C01819=1087.779,-102.417,-50.994,174.374,16.859,152.716
C01820=1087.774,-102.667,-50.984,174.373,16.858,152.716
C01821=1087.768,-102.917,-50.974,174.371,16.857,152.716
C01822=1087.761,-103.166,-50.965,174.369,16.856,152.716
C01823=1087.755,-103.416,-50.955,174.368,16.856,152.716
C01824=1087.749,-103.666,-50.944,174.367,16.855,152.716
C01825=1087.743,-103.916,-50.935,174.365,16.854,152.716
C01826=1087.737,-104.165,-50.925,174.363,16.853,152.717
C01827=1087.731,-104.415,-50.915,174.362,16.852,152.717
C01828=1087.724,-104.664,-50.905,174.361,16.851,152.717
C01829=1087.719,-104.914,-50.895,174.359,16.851,152.717
C01830=1087.713,-105.164,-50.886,174.357,16.850,152.717
C01831=1087.707,-105.414,-50.876,174.355,16.849,152.717
C01832=1087.700,-105.663,-50.866,174.354,16.849,152.718
C01833=1087.695,-105.913,-50.856,174.353,16.847,152.718
C01834=1087.689,-106.163,-50.846,174.351,16.847,152.718
C01835=1087.682,-106.413,-50.837,174.349,16.846,152.718
C01836=1087.676,-106.663,-50.827,174.348,16.845,152.718
C01837=1087.670,-106.912,-50.817,174.347,16.845,152.718
C01838=1087.664,-107.162,-50.807,174.345,16.844,152.718
C01839=1087.658,-107.412,-50.797,174.343,16.842,152.719
C01840=1087.652,-107.662,-50.787,174.342,16.842,152.719
C01841=1087.646,-107.911,-50.778,174.341,16.841,152.719
C01842=1087.640,-108.161,-50.768,174.339,16.841,152.719
C01843=1087.633,-108.411,-50.759,174.337,16.840,152.719
C01844=1087.627,-108.660,-50.748,174.336,16.840,152.719
C01845=1087.621,-108.910,-50.739,174.334,16.839,152.720
C01846=1087.615,-109.160,-50.729,174.333,16.837,152.720
C01847=1087.609,-109.410,-50.719,174.331,16.837,152.720
C01848=1087.603,-109.660,-50.710,174.330,16.836,152.720
C01849=1087.597,-109.909,-50.700,174.328,16.836,152.720
C01850=1087.591,-110.159,-50.691,174.326,16.835,152.720
C01851=1087.585,-110.408,-50.681,174.324,16.834,152.721
C01852=1087.579,-110.658,-50.672,174.324,16.833,152.721
C01853=1087.573,-110.908,-50.662,174.322,16.833,152.721
C01854=1087.567,-111.158,-50.653,174.320,16.832,152.721
C01855=1087.560,-111.407,-50.642,174.318,16.831,152.721
C01856=1087.554,-111.657,-50.633,174.317,16.831,152.721
C01857=1087.548,-111.907,-50.623,174.315,16.830,152.722
C01858=1087.542,-112.156,-50.614,174.314,16.829,152.722
C01859=1087.535,-112.406,-50.604,174.313,16.829,152.722
C01860=1087.529,-112.656,-50.594,174.311,16.828,152.722
C01861=1087.523,-112.927,-50.584,174.309,16.827,152.722
C01862=1087.517,-113.198,-50.574,174.307,16.826,152.723
C01863=1087.510,-113.469,-50.563,174.306,16.826,152.723
C01864=1087.503,-113.741,-50.553,174.304,16.824,152.723
C01865=1087.497,-113.991,-50.543,174.303,16.824,152.723
C01866=1087.491,-114.240,-50.534,174.301,16.823,152.723
C01867=1087.485,-114.490,-50.524,174.299,16.823,152.724
C01868=1087.479,-114.740,-50.515,174.298,16.822,152.724
C01869=1087.473,-114.989,-50.505,174.296,16.822,152.724
C01870=1087.467,-115.239,-50.496,174.295,16.821,152.724
C01871=1087.461,-115.489,-50.486,174.293,16.820,152.724
C01872=1087.454,-115.738,-50.477,174.292,16.819,152.724
C01873=1087.448,-115.988,-50.467,174.290,16.819,152.725
C01874=1087.442,-116.238,-50.458,174.288,16.818,152.725
C01875=1087.436,-116.488,-50.448,174.287,16.818,152.725
C01876=1087.430,-116.738,-50.438,174.286,16.817,152.725
C01877=1087.424,-116.987,-50.429,174.284,16.816,152.725
C01878=1087.418,-117.238,-50.420,174.282,16.815,152.726
C01879=1087.412,-117.487,-50.411,174.281,16.815,152.726
C01880=1087.406,-117.737,-50.401,174.279,16.814,152.726
C01881=1087.399,-117.986,-50.392,174.277,16.814,152.726
C01882=1087.393,-118.236,-50.383,174.276,16.813,152.726
C01883=1087.387,-118.486,-50.373,174.275,16.813,152.726
C01884=1087.381,-118.736,-50.364,174.273,16.812,152.727
C01885=1087.374,-118.985,-50.354,174.272,16.811,152.727
C01886=1087.368,-119.235,-50.344,174.270,16.811,152.727
C01887=1087.363,-119.484,-50.335,174.268,16.810,152.727
C01888=1087.357,-119.735,-50.326,174.267,16.810,152.727
C01889=1087.351,-119.985,-50.317,174.265,16.809,152.728
C01890=1087.344,-120.234,-50.308,174.264,16.808,152.728
C01891=1087.338,-120.484,-50.298,174.262,16.808,152.728
C01892=1087.331,-120.734,-50.289,174.261,16.807,152.728
C01893=1087.325,-120.983,-50.279,174.259,16.806,152.728
C01894=1087.320,-121.233,-50.271,174.257,16.806,152.729
C01895=1087.314,-121.483,-50.261,174.256,16.806,152.729
C01896=1087.308,-121.733,-50.252,174.254,16.805,152.729
C01897=1087.301,-121.982,-50.243,174.252,16.804,152.729
C01898=1087.295,-122.232,-50.233,174.251,16.804,152.729
C01899=1087.288,-122.482,-50.223,174.250,16.803,152.730
C01900=1087.283,-122.732,-50.215,174.248,16.802,152.730
C01901=1087.277,-122.981,-50.205,174.247,16.802,152.730
C01902=1087.271,-123.231,-50.196,174.245,16.801,152.730
C01903=1087.264,-123.481,-50.187,174.243,16.801,152.730
C01904=1087.258,-123.731,-50.178,174.242,16.801,152.731
C01905=1087.252,-123.981,-50.168,174.240,16.800,152.731
C01906=1087.246,-124.230,-50.159,174.238,16.799,152.731
C01907=1087.240,-124.480,-50.150,174.237,16.799,152.731
C01908=1087.234,-124.730,-50.141,174.236,16.798,152.731
C01909=1087.227,-124.980,-50.132,174.234,16.797,152.732
C01910=1087.221,-125.229,-50.122,174.233,16.797,152.732
C01911=1087.216,-125.479,-50.113,174.231,16.797,152.732
C01912=1087.209,-125.729,-50.105,174.229,16.796,152.732
C01913=1087.203,-125.978,-50.095,174.228,16.796,152.732
C01914=1087.197,-126.228,-50.086,174.226,16.795,152.733
C01915=1087.190,-126.478,-50.076,174.225,16.795,152.733
C01916=1087.184,-126.728,-50.068,174.223,16.794,152.733
C01917=1087.178,-126.977,-50.059,174.221,16.793,152.733
C01918=1087.172,-127.227,-50.049,174.220,16.793,152.734
C01919=1087.165,-127.477,-50.041,174.218,16.793,152.734
C01920=1087.159,-127.727,-50.031,174.216,16.792,152.734
C01921=1087.153,-127.984,-50.022,174.215,16.792,152.734
C01922=1087.148,-128.242,-50.012,174.214,16.790,152.734
C01923=1087.150,-128.498,-50.000,174.213,16.788,152.734
C01924=1087.156,-128.753,-49.987,174.213,16.784,152.733
C01925=1086.753,-128.774,-50.114,174.170,16.892,152.762
C01926=1086.746,-128.521,-50.128,174.171,16.896,152.763
C01927=1086.745,-128.264,-50.139,174.172,16.899,152.763
C01928=1086.750,-128.006,-50.150,174.173,16.900,152.763
C01929=1086.756,-127.749,-50.159,174.175,16.900,152.763
C01930=1086.762,-127.499,-50.167,174.177,16.901,152.763
C01931=1086.768,-127.249,-50.177,174.178,16.901,152.762
C01932=1086.774,-126.999,-50.187,174.180,16.902,152.762
C01933=1086.780,-126.750,-50.194,174.181,16.903,152.762
C01934=1086.786,-126.500,-50.204,174.182,16.903,152.762
C01935=1086.792,-126.250,-50.214,174.184,16.904,152.762
C01936=1086.799,-126.000,-50.222,174.186,16.904,152.761
C01937=1086.805,-125.750,-50.231,174.187,16.904,152.761
C01938=1086.811,-125.501,-50.241,174.189,16.905,152.761
C01939=1086.817,-125.252,-50.250,174.191,16.906,152.761
C01940=1086.823,-125.001,-50.258,174.192,16.906,152.760
C01941=1086.830,-124.752,-50.268,174.194,16.907,152.760
C01942=1086.836,-124.502,-50.278,174.195,16.908,152.760
C01943=1086.842,-124.252,-50.287,174.197,16.908,152.760
C01944=1086.847,-124.002,-50.296,174.198,16.909,152.760
C01945=1086.854,-123.753,-50.305,174.200,16.909,152.760
C01946=1086.860,-123.503,-50.314,174.201,16.909,152.759
C01947=1086.866,-123.253,-50.324,174.203,16.910,152.759
C01948=1086.873,-123.003,-50.333,174.205,16.911,152.759
C01949=1086.878,-122.754,-50.342,174.206,16.911,152.759
C01950=1086.885,-122.504,-50.351,174.208,16.912,152.759
C01951=1086.891,-122.254,-50.360,174.209,16.913,152.758
C01952=1086.897,-122.005,-50.370,174.211,16.913,152.758
C01953=1086.903,-121.755,-50.379,174.212,16.914,152.758
C01954=1086.909,-121.504,-50.388,174.214,16.914,152.758
C01955=1086.915,-121.255,-50.398,174.215,16.914,152.758
C01956=1086.921,-121.005,-50.407,174.217,16.915,152.757
C01957=1086.928,-120.756,-50.416,174.219,16.916,152.757
C01958=1086.934,-120.506,-50.426,174.220,16.917,152.757
C01959=1086.940,-120.256,-50.435,174.222,16.917,152.757
C01960=1086.946,-120.006,-50.444,174.223,16.918,152.757
C01961=1086.952,-119.756,-50.454,174.224,16.918,152.756
C01962=1086.958,-119.507,-50.463,174.226,16.919,152.756
C01963=1086.964,-119.257,-50.472,174.228,16.920,152.756
C01964=1086.970,-119.008,-50.482,174.230,16.921,152.756
C01965=1086.977,-118.758,-50.491,174.231,16.921,152.756
C01966=1086.983,-118.508,-50.500,174.232,16.922,152.755
C01967=1086.989,-118.258,-50.510,174.234,16.922,152.755
C01968=1086.995,-118.008,-50.519,174.235,16.923,152.755
C01969=1087.001,-117.758,-50.528,174.237,16.923,152.755
C01970=1087.007,-117.509,-50.538,174.239,16.924,152.755
C01971=1087.013,-117.259,-50.547,174.240,16.924,152.755
C01972=1087.019,-117.010,-50.557,174.242,16.925,152.754
C01973=1087.025,-116.760,-50.566,174.243,16.926,152.754
C01974=1087.032,-116.510,-50.576,174.245,16.927,152.754
C01975=1087.038,-116.260,-50.586,174.246,16.927,152.754
C01976=1087.044,-116.010,-50.595,174.248,16.928,152.754
C01977=1087.050,-115.761,-50.605,174.250,16.929,152.753
C01978=1087.056,-115.511,-50.614,174.251,16.929,152.753
C01979=1087.062,-115.262,-50.623,174.253,16.930,152.753
C01980=1087.069,-115.012,-50.632,174.254,16.931,152.753
C01981=1087.075,-114.762,-50.642,174.256,16.932,152.753
C01982=1087.081,-114.513,-50.652,174.257,16.932,152.753
C01983=1087.087,-114.263,-50.661,174.259,16.933,152.752
C01984=1087.094,-114.013,-50.671,174.261,16.933,152.752
C01985=1087.099,-113.763,-50.681,174.262,16.934,152.752
C01986=1087.106,-113.491,-50.691,174.263,16.935,152.752
C01987=1087.112,-113.220,-50.701,174.265,16.936,152.752
C01988=1087.119,-112.948,-50.712,174.267,16.936,152.751
C01989=1087.125,-112.677,-50.722,174.269,16.937,152.751
C01990=1087.131,-112.427,-50.732,174.271,16.938,152.751
C01991=1087.138,-112.177,-50.741,174.271,16.938,152.751
C01992=1087.144,-111.927,-50.751,174.273,16.939,152.751
C01993=1087.150,-111.677,-50.760,174.275,16.940,152.751
C01994=1087.156,-111.428,-50.770,174.277,16.941,152.750
C01995=1087.162,-111.178,-50.779,174.278,16.941,152.750
C01996=1087.168,-110.928,-50.789,174.279,16.942,152.750
C01997=1087.174,-110.680,-50.799,174.281,16.943,152.750
C01998=1087.181,-110.430,-50.808,174.283,16.944,152.750
C01999=1087.187,-110.180,-50.818,174.284,16.944,152.750
C02000=1087.193,-109.930,-50.828,174.286,16.945,152.749
C02001=1087.199,-109.680,-50.837,174.288,16.946,152.749
C02002=1087.205,-109.431,-50.847,174.289,16.947,152.749
C02003=1087.211,-109.180,-50.857,174.290,16.947,152.749
C02004=1087.217,-108.931,-50.866,174.292,16.948,152.749
C02005=1087.223,-108.681,-50.876,174.294,16.949,152.749
C02006=1087.229,-108.431,-50.886,174.296,16.950,152.748
C02007=1087.236,-108.182,-50.896,174.296,16.950,152.748
C02008=1087.242,-107.932,-50.905,174.298,16.951,152.748
C02009=1087.248,-107.682,-50.915,174.300,16.952,152.748
C02010=1087.254,-107.433,-50.925,174.302,16.953,152.748
C02011=1087.260,-107.183,-50.934,174.302,16.953,152.748
C02012=1087.266,-106.933,-50.944,174.304,16.954,152.748
C02013=1087.272,-106.683,-50.955,174.306,16.955,152.747
C02014=1087.278,-106.434,-50.964,174.308,16.956,152.747
C02015=1087.285,-106.184,-50.974,174.309,16.956,152.747
C02016=1087.291,-105.934,-50.983,174.310,16.957,152.747
C02017=1087.296,-105.684,-50.993,174.312,16.958,152.747
C02018=1087.302,-105.434,-51.003,174.314,16.959,152.747
C02019=1087.309,-105.185,-51.013,174.315,16.960,152.746
C02020=1087.315,-104.935,-51.023,174.316,16.961,152.746
C02021=1087.321,-104.685,-51.032,174.318,16.961,152.746
C02022=1087.327,-104.435,-51.043,174.320,16.962,152.746
C02023=1087.333,-104.185,-51.052,174.321,16.963,152.746
C02024=1087.339,-103.936,-51.062,174.323,16.963,152.746
C02025=1087.345,-103.686,-51.072,174.324,16.964,152.746
C02026=1087.351,-103.436,-51.082,174.326,16.966,152.745
C02027=1087.357,-103.187,-51.092,174.328,16.967,152.745
C02028=1087.364,-102.937,-51.102,174.329,16.967,152.745
C02029=1087.370,-102.688,-51.112,174.330,16.968,152.745
C02030=1087.375,-102.437,-51.122,174.332,16.969,152.745
C02031=1087.382,-102.188,-51.132,174.334,16.969,152.745
C02032=1087.388,-101.938,-51.142,174.335,16.971,152.745
C02033=1087.394,-101.689,-51.151,174.337,16.972,152.744
C02034=1087.399,-101.439,-51.161,174.338,16.972,152.744
C02035=1087.406,-101.189,-51.172,174.340,16.973,152.744
C02036=1087.412,-100.940,-51.181,174.341,16.974,152.744
C02037=1087.417,-100.690,-51.191,174.343,16.975,152.744
C02038=1087.424,-100.440,-51.202,174.345,16.976,152.744
C02039=1087.430,-100.191,-51.211,174.346,16.976,152.744
C02040=1087.436,-99.941,-51.221,174.347,16.977,152.743
C02041=1087.442,-99.691,-51.232,174.349,16.978,152.743
C02042=1087.448,-99.441,-51.241,174.351,16.979,152.743
C02043=1087.454,-99.192,-51.251,174.353,16.980,152.743
C02044=1087.460,-98.942,-51.262,174.353,16.980,152.743
C02045=1087.467,-98.692,-51.272,174.355,16.982,152.743
C02046=1087.473,-98.442,-51.281,174.357,16.983,152.743
C02047=1087.479,-98.192,-51.292,174.358,16.984,152.743
C02048=1087.485,-97.943,-51.302,174.360,16.984,152.742
C02049=1087.491,-97.693,-51.312,174.361,16.985,152.742
C02050=1087.498,-97.416,-51.323,174.363,16.986,152.742
C02051=1087.504,-97.139,-51.334,174.364,16.987,152.742
C02052=1087.511,-96.863,-51.346,174.366,16.988,152.742
C02053=1087.517,-96.586,-51.356,174.368,16.989,152.742
C02054=1087.523,-96.336,-51.367,174.370,16.990,152.742
C02055=1087.529,-96.087,-51.377,174.371,16.991,152.741
C02056=1087.535,-95.837,-51.386,174.373,16.992,152.741
C02057=1087.541,-95.587,-51.397,174.375,16.993,152.741
C02058=1087.548,-95.337,-51.407,174.376,16.994,152.741
C02059=1087.554,-95.087,-51.418,174.377,16.995,152.741
C02060=1087.560,-94.838,-51.428,174.379,16.996,152.741
C02061=1087.565,-94.588,-51.438,174.380,16.997,152.741
C02062=1087.572,-94.338,-51.448,174.382,16.998,152.741
C02063=1087.577,-94.088,-51.458,174.384,16.999,152.741
C02064=1087.584,-93.839,-51.469,174.385,17.000,152.740
C02065=1087.589,-93.589,-51.479,174.386,17.000,152.740
C02066=1087.596,-93.340,-51.489,174.388,17.001,152.740
C02067=1087.601,-93.090,-51.499,174.390,17.002,152.740
C02068=1087.607,-92.841,-51.509,174.391,17.004,152.740
C02069=1087.613,-92.590,-51.520,174.393,17.005,152.740
C02070=1087.619,-92.341,-51.531,174.394,17.006,152.740
C02071=1087.625,-92.090,-51.540,174.396,17.007,152.740
C02072=1087.631,-91.841,-51.551,174.397,17.007,152.740
C02073=1087.637,-91.591,-51.561,174.399,17.008,152.739
C02074=1087.643,-91.342,-51.572,174.400,17.010,152.739
C02075=1087.649,-91.092,-51.581,174.402,17.011,152.739
C02076=1087.655,-90.842,-51.592,174.403,17.012,152.739
C02077=1087.661,-90.593,-51.602,174.405,17.013,152.739
C02078=1087.667,-90.343,-51.613,174.407,17.013,152.739
C02079=1087.674,-90.093,-51.623,174.408,17.014,152.739
C02080=1087.679,-89.843,-51.633,174.410,17.015,152.739
C02081=1087.686,-89.594,-51.644,174.411,17.016,152.738
C02082=1087.691,-89.344,-51.654,174.413,17.017,152.738
C02083=1087.697,-89.094,-51.665,174.414,17.018,152.738
C02084=1087.704,-88.845,-51.675,174.416,17.019,152.738
C02085=1087.709,-88.595,-51.685,174.418,17.021,152.738
C02086=1087.716,-88.345,-51.696,174.419,17.021,152.738
C02087=1087.721,-88.095,-51.706,174.420,17.022,152.738
C02088=1087.728,-87.846,-51.716,174.422,17.023,152.738
C02089=1087.734,-87.596,-51.727,174.423,17.024,152.738
C02090=1087.739,-87.346,-51.737,174.425,17.025,152.737
C02091=1087.746,-87.097,-51.748,174.427,17.027,152.737
C02092=1087.752,-86.847,-51.759,174.428,17.028,152.737
C02093=1087.758,-86.597,-51.768,174.430,17.029,152.737
C02094=1087.764,-86.348,-51.779,174.431,17.029,152.737
C02095=1087.770,-86.098,-51.790,174.432,17.030,152.737
C02096=1087.776,-85.848,-51.800,174.434,17.031,152.737
C02097=1087.782,-85.598,-51.811,174.436,17.033,152.737
C02098=1087.789,-85.349,-51.821,174.437,17.034,152.737
C02099=1087.794,-85.099,-51.831,174.439,17.035,152.737
C02100=1087.800,-84.849,-51.842,174.441,17.036,152.736
C02101=1087.806,-84.600,-51.853,174.442,17.037,152.736
C02102=1087.813,-84.350,-51.864,174.443,17.037,152.736
C02103=1087.819,-84.100,-51.873,174.445,17.039,152.736
C02104=1087.824,-83.851,-51.884,174.446,17.040,152.736
C02105=1087.830,-83.601,-51.895,174.448,17.041,152.736
C02106=1087.837,-83.351,-51.905,174.450,17.042,152.736
C02107=1087.843,-83.101,-51.916,174.451,17.043,152.736
C02108=1087.849,-82.852,-51.926,174.453,17.044,152.736
C02109=1087.855,-82.603,-51.937,174.455,17.045,152.735
C02110=1087.861,-82.352,-51.948,174.456,17.046,152.735
C02111=1087.867,-82.103,-51.958,174.457,17.047,152.735
C02112=1087.873,-81.853,-51.969,174.459,17.048,152.735
C02113=1087.879,-81.604,-51.980,174.460,17.049,152.735
C02114=1087.886,-81.329,-51.991,174.462,17.050,152.735
C02115=1087.893,-81.054,-52.003,174.464,17.051,152.735
C02116=1087.899,-80.779,-52.015,174.466,17.053,152.735
C02117=1087.906,-80.505,-52.026,174.467,17.054,152.735
C02118=1087.913,-80.255,-52.037,174.469,17.055,152.735
C02119=1087.918,-80.005,-52.048,174.470,17.056,152.735
C02120=1087.924,-79.756,-52.059,174.472,17.057,152.734
C02121=1087.931,-79.507,-52.069,174.473,17.058,152.734
C02122=1087.937,-79.257,-52.080,174.475,17.059,152.734
C02123=1087.942,-79.006,-52.090,174.476,17.060,152.734
C02124=1087.948,-78.757,-52.101,174.478,17.061,152.734
C02125=1087.954,-78.507,-52.112,174.480,17.063,152.734
C02126=1087.961,-78.258,-52.123,174.481,17.064,152.734
C02127=1087.967,-78.008,-52.134,174.483,17.065,152.734
C02128=1087.972,-77.759,-52.145,174.484,17.066,152.734
C02129=1087.978,-77.509,-52.155,174.486,17.067,152.734
C02130=1087.984,-77.259,-52.167,174.488,17.069,152.733
C02131=1087.990,-77.009,-52.177,174.489,17.070,152.733
C02132=1087.996,-76.759,-52.188,174.490,17.070,152.733
C02133=1088.002,-76.510,-52.198,174.491,17.072,152.733
C02134=1088.008,-76.260,-52.209,174.493,17.073,152.733
C02135=1088.014,-76.010,-52.220,174.495,17.074,152.733
C02136=1088.020,-75.761,-52.231,174.496,17.075,152.733
C02137=1088.026,-75.512,-52.242,174.498,17.076,152.733
C02138=1088.032,-75.261,-52.253,174.500,17.077,152.733
C02139=1088.038,-75.012,-52.263,174.501,17.079,152.733
C02140=1088.044,-74.763,-52.274,174.503,17.080,152.733
C02141=1088.051,-74.512,-52.285,174.504,17.081,152.733
C02142=1088.056,-74.263,-52.296,174.506,17.082,152.733
C02143=1088.062,-74.013,-52.307,174.508,17.083,152.732
C02144=1088.068,-73.763,-52.318,174.509,17.085,152.732
C02145=1088.074,-73.514,-52.329,174.511,17.086,152.732
C02146=1088.080,-73.264,-52.340,174.512,17.087,152.732
C02147=1088.086,-73.015,-52.351,174.514,17.088,152.732
C02148=1088.092,-72.765,-52.362,174.515,17.090,152.732
C02149=1088.098,-72.515,-52.373,174.517,17.091,152.732
C02150=1088.103,-72.266,-52.384,174.518,17.091,152.732
C02151=1088.109,-72.016,-52.395,174.519,17.093,152.732
C02152=1088.115,-71.766,-52.406,174.521,17.094,152.732
C02153=1088.121,-71.516,-52.417,174.522,17.095,152.732
C02154=1088.126,-71.267,-52.429,174.524,17.096,152.732
C02155=1088.132,-71.017,-52.439,174.525,17.098,152.732
C02156=1088.138,-70.767,-52.451,174.527,17.099,152.732
C02157=1088.144,-70.518,-52.462,174.529,17.100,152.732
C02158=1088.150,-70.268,-52.472,174.530,17.102,152.732
C02159=1088.156,-70.018,-52.484,174.532,17.103,152.731
C02160=1088.162,-69.768,-52.495,174.533,17.104,152.731
C02161=1088.168,-69.519,-52.505,174.535,17.105,152.731
C02162=1088.174,-69.269,-52.517,174.536,17.107,152.731
C02163=1088.180,-69.019,-52.528,174.538,17.108,152.731
C02164=1088.186,-68.770,-52.539,174.539,17.109,152.731
C02165=1088.192,-68.520,-52.550,174.541,17.110,152.731
C02166=1088.197,-68.270,-52.562,174.542,17.111,152.731
C02167=1088.203,-68.021,-52.573,174.544,17.113,152.731
C02168=1088.209,-67.771,-52.584,174.545,17.114,152.731
C02169=1088.215,-67.521,-52.595,174.547,17.115,152.731
C02170=1088.221,-67.272,-52.606,174.549,17.116,152.731
C02171=1088.227,-67.021,-52.617,174.550,17.118,152.731
C02172=1088.233,-66.773,-52.629,174.552,17.119,152.731
C02173=1088.239,-66.523,-52.639,174.553,17.120,152.731
C02174=1088.245,-66.273,-52.651,174.555,17.122,152.731
C02175=1088.250,-66.023,-52.662,174.556,17.123,152.730
C02176=1088.256,-65.774,-52.673,174.558,17.124,152.730
C02177=1088.262,-65.524,-52.685,174.559,17.126,152.730
C02178=1088.269,-65.251,-52.696,174.561,17.127,152.730
C02179=1088.275,-64.979,-52.709,174.563,17.128,152.730
C02180=1088.282,-64.707,-52.721,174.564,17.129,152.730
C02181=1088.288,-64.434,-52.734,174.566,17.131,152.730
C02182=1088.294,-64.185,-52.745,174.567,17.131,152.730
C02183=1088.300,-63.935,-52.756,174.569,17.133,152.730
C02184=1088.306,-63.686,-52.767,174.570,17.134,152.730
C02185=1088.311,-63.436,-52.779,174.572,17.135,152.730
C02186=1088.318,-63.186,-52.790,174.573,17.137,152.730
C02187=1088.323,-62.936,-52.801,174.575,17.138,152.730
C02188=1088.330,-62.687,-52.813,174.577,17.139,152.730
C02189=1088.336,-62.437,-52.824,174.578,17.141,152.730
C02190=1088.342,-62.188,-52.835,174.580,17.142,152.730
C02191=1088.347,-61.938,-52.847,174.582,17.143,152.729
C02192=1088.353,-61.688,-52.858,174.583,17.145,152.730
C02193=1088.360,-61.438,-52.869,174.585,17.146,152.729
C02194=1088.366,-61.189,-52.881,174.587,17.147,152.729
C02195=1088.372,-60.939,-52.892,174.588,17.149,152.729
C02196=1088.378,-60.690,-52.903,174.590,17.150,152.729
C02197=1088.383,-60.439,-52.915,174.591,17.152,152.729
C02198=1088.389,-60.190,-52.927,174.593,17.153,152.729
C02199=1088.396,-59.940,-52.938,174.594,17.154,152.729
C02200=1088.402,-59.691,-52.949,174.596,17.155,152.729
C02201=1088.407,-59.442,-52.960,174.597,17.156,152.729
C02202=1088.413,-59.191,-52.972,174.599,17.157,152.729
C02203=1088.419,-58.942,-52.984,174.600,17.159,152.729
C02204=1088.425,-58.692,-52.995,174.602,17.160,152.729
C02205=1088.431,-58.443,-53.006,174.604,17.161,152.729
C02206=1088.437,-58.193,-53.018,174.605,17.163,152.729
C02207=1088.443,-57.943,-53.029,174.607,17.164,152.729
C02208=1088.449,-57.694,-53.041,174.608,17.166,152.729
C02209=1088.455,-57.444,-53.052,174.610,17.167,152.729
C02210=1088.462,-57.194,-53.063,174.611,17.168,152.728
C02211=1088.467,-56.945,-53.076,174.613,17.169,152.729
C02212=1088.473,-56.695,-53.087,174.614,17.170,152.728
C02213=1088.480,-56.445,-53.099,174.616,17.172,152.728
C02214=1088.486,-56.196,-53.110,174.617,17.173,152.728
C02215=1088.492,-55.946,-53.122,174.619,17.174,152.728
C02216=1088.497,-55.696,-53.133,174.620,17.176,152.728
C02217=1088.504,-55.447,-53.145,174.622,17.177,152.728
C02218=1088.510,-55.197,-53.156,174.623,17.178,152.728
C02219=1088.516,-54.947,-53.168,174.625,17.180,152.728
C02220=1088.521,-54.698,-53.179,174.626,17.181,152.728
C02221=1088.528,-54.448,-53.191,174.628,17.182,152.728
C02222=1088.533,-54.198,-53.203,174.629,17.183,152.728
C02223=1088.540,-53.949,-53.215,174.631,17.185,152.728
C02224=1088.546,-53.699,-53.226,174.632,17.186,152.728
C02225=1088.552,-53.450,-53.238,174.634,17.187,152.728
C02226=1088.558,-53.199,-53.249,174.636,17.188,152.728
C02227=1088.564,-52.950,-53.261,174.637,17.190,152.728
C02228=1088.570,-52.700,-53.272,174.639,17.191,152.728
C02229=1088.576,-52.451,-53.284,174.641,17.193,152.728
C02230=1088.582,-52.201,-53.296,174.643,17.194,152.728
C02231=1088.588,-51.951,-53.308,174.644,17.195,152.727
C02232=1088.594,-51.702,-53.319,174.646,17.197,152.727
C02233=1088.600,-51.452,-53.331,174.647,17.198,152.727
C02234=1088.607,-51.202,-53.343,174.649,17.200,152.727
C02235=1088.612,-50.953,-53.354,174.650,17.201,152.727
C02236=1088.618,-50.703,-53.366,174.652,17.202,152.727
C02237=1088.624,-50.453,-53.377,174.653,17.203,152.727
C02238=1088.631,-50.204,-53.389,174.655,17.205,152.727
C02239=1088.636,-49.955,-53.401,174.656,17.206,152.727
C02240=1088.641,-49.704,-53.413,174.658,17.207,152.727
C02241=1088.648,-49.455,-53.425,174.659,17.209,152.727
C02242=1088.654,-49.184,-53.438,174.661,17.210,152.727
C02243=1088.660,-48.913,-53.451,174.663,17.212,152.727
C02244=1088.667,-48.641,-53.464,174.664,17.214,152.727
C02245=1088.673,-48.371,-53.476,174.666,17.215,152.727
C02246=1088.679,-48.121,-53.489,174.667,17.216,152.727
C02247=1088.686,-47.871,-53.501,174.669,17.217,152.727
C02248=1088.691,-47.621,-53.512,174.670,17.219,152.727
C02249=1088.697,-47.372,-53.524,174.673,17.221,152.727
C02250=1088.703,-47.123,-53.536,174.674,17.222,152.727
C02251=1088.708,-46.872,-53.548,174.676,17.223,152.727
C02252=1088.714,-46.623,-53.560,174.677,17.225,152.727
C02253=1088.720,-46.373,-53.572,174.679,17.226,152.727
C02254=1088.727,-46.123,-53.584,174.680,17.228,152.727
C02255=1088.732,-45.874,-53.596,174.682,17.229,152.727
C02256=1088.738,-45.625,-53.608,174.683,17.230,152.727
C02257=1088.744,-45.375,-53.620,174.685,17.232,152.727
C02258=1088.749,-45.125,-53.632,174.686,17.233,152.727
C02259=1088.756,-44.875,-53.644,174.688,17.235,152.727
C02260=1088.761,-44.626,-53.656,174.689,17.236,152.727
C02261=1088.768,-44.377,-53.668,174.691,17.238,152.726
C02262=1088.774,-44.126,-53.680,174.693,17.239,152.726
C02263=1088.779,-43.877,-53.692,174.694,17.241,152.726
C02264=1088.786,-43.627,-53.704,174.696,17.242,152.726
C02265=1088.791,-43.378,-53.716,174.697,17.243,152.726
C02266=1088.797,-43.128,-53.727,174.699,17.244,152.726
C02267=1088.803,-42.878,-53.740,174.700,17.246,152.726
C02268=1088.808,-42.629,-53.752,174.702,17.247,152.726
C02269=1088.815,-42.379,-53.764,174.703,17.249,152.726
C02270=1088.821,-42.129,-53.776,174.705,17.250,152.726
C02271=1088.826,-41.880,-53.789,174.706,17.251,152.726
C02272=1088.833,-41.630,-53.800,174.709,17.254,152.726
C02273=1088.838,-41.380,-53.812,174.710,17.255,152.726
C02274=1088.845,-41.131,-53.824,174.712,17.256,152.726
C02275=1088.850,-40.881,-53.837,174.713,17.257,152.726
C02276=1088.856,-40.631,-53.849,174.715,17.259,152.726
C02277=1088.862,-40.383,-53.861,174.716,17.260,152.726
C02278=1088.868,-40.133,-53.873,174.718,17.262,152.726
C02279=1088.874,-39.883,-53.886,174.719,17.263,152.726
C02280=1088.881,-39.633,-53.897,174.721,17.264,152.726
C02281=1088.886,-39.383,-53.909,174.723,17.266,152.726
C02282=1088.892,-39.134,-53.922,174.724,17.268,152.726
C02283=1088.898,-38.884,-53.934,174.726,17.269,152.726
C02284=1088.904,-38.635,-53.946,174.728,17.270,152.726
C02285=1088.910,-38.385,-53.959,174.729,17.272,152.726
C02286=1088.916,-38.135,-53.971,174.731,17.273,152.726
C02287=1088.922,-37.886,-53.983,174.732,17.275,152.726
C02288=1088.928,-37.636,-53.995,174.733,17.276,152.726
C02289=1088.933,-37.386,-54.008,174.735,17.277,152.726
C02290=1088.939,-37.137,-54.020,174.737,17.279,152.726
C02291=1088.945,-36.887,-54.033,174.738,17.281,152.726
C02292=1088.951,-36.637,-54.045,174.740,17.282,152.726
C02293=1088.957,-36.388,-54.057,174.741,17.284,152.726
C02294=1088.962,-36.139,-54.069,174.743,17.285,152.726
C02295=1088.968,-35.889,-54.082,174.744,17.286,152.726
C02296=1088.974,-35.639,-54.094,174.746,17.288,152.726
C02297=1088.980,-35.390,-54.107,174.747,17.289,152.726
C02298=1088.986,-35.140,-54.119,174.750,17.291,152.726
C02299=1088.991,-34.890,-54.132,174.751,17.292,152.725
C02300=1088.998,-34.640,-54.144,174.753,17.294,152.726
C02301=1089.003,-34.391,-54.156,174.754,17.295,152.726
C02302=1089.009,-34.141,-54.168,174.756,17.297,152.725
C02303=1089.015,-33.891,-54.181,174.757,17.298,152.726
C02304=1089.021,-33.642,-54.193,174.758,17.300,152.726
C02305=1089.026,-33.392,-54.206,174.761,17.301,152.725
C02306=1089.034,-33.122,-54.219,174.762,17.303,152.725
C02307=1089.039,-32.851,-54.232,174.764,17.305,152.726
C02308=1089.046,-32.580,-54.246,174.765,17.306,152.725
C02309=1089.052,-32.309,-54.260,174.767,17.308,152.725
C02310=1089.058,-32.060,-54.272,174.769,17.309,152.725
C02311=1089.064,-31.810,-54.285,174.770,17.311,152.725
C02312=1089.069,-31.561,-54.297,174.772,17.312,152.725
C02313=1089.076,-31.311,-54.309,174.773,17.313,152.725
C02314=1089.082,-31.062,-54.322,174.776,17.315,152.725
C02315=1089.088,-30.812,-54.335,174.777,17.317,152.725
C02316=1089.094,-30.562,-54.347,174.779,17.318,152.725
C02317=1089.099,-30.313,-54.359,174.780,17.320,152.725
C02318=1089.105,-30.063,-54.372,174.782,17.321,152.725
C02319=1089.111,-29.813,-54.385,174.783,17.322,152.725
C02320=1089.117,-29.564,-54.398,174.784,17.324,152.725
C02321=1089.123,-29.314,-54.410,174.787,17.326,152.725
C02322=1089.129,-29.065,-54.423,174.788,17.327,152.725
C02323=1089.134,-28.815,-54.435,174.790,17.329,152.725
C02324=1089.140,-28.565,-54.448,174.791,17.330,152.725
C02325=1089.147,-28.316,-54.460,174.793,17.331,152.725
C02326=1089.153,-28.066,-54.473,174.794,17.333,152.725
C02327=1089.159,-27.816,-54.485,174.796,17.334,152.725
C02328=1089.164,-27.567,-54.498,174.798,17.336,152.725
C02329=1089.170,-27.317,-54.510,174.799,17.337,152.725
C02330=1089.177,-27.068,-54.523,174.801,17.339,152.725
C02331=1089.182,-26.818,-54.536,174.802,17.341,152.725
C02332=1089.188,-26.568,-54.549,174.804,17.342,152.725
C02333=1089.195,-26.319,-54.562,174.805,17.343,152.725
C02334=1089.199,-26.069,-54.575,174.807,17.345,152.725
C02335=1089.205,-25.819,-54.587,174.809,17.347,152.725
C02336=1089.211,-25.570,-54.600,174.810,17.348,152.725
C02337=1089.217,-25.320,-54.613,174.812,17.350,152.725
C02338=1089.223,-25.070,-54.626,174.813,17.351,152.725
C02339=1089.228,-24.821,-54.638,174.815,17.352,152.725
C02340=1089.235,-24.572,-54.651,174.817,17.355,152.725
C02341=1089.240,-24.322,-54.664,174.818,17.356,152.725
C02342=1089.246,-24.072,-54.676,174.820,17.357,152.725
C02343=1089.252,-23.823,-54.690,174.821,17.359,152.725
C02344=1089.258,-23.573,-54.702,174.823,17.360,152.725
C02345=1089.263,-23.324,-54.715,174.825,17.362,152.725
C02346=1089.269,-23.074,-54.728,174.826,17.364,152.725
C02347=1089.275,-22.824,-54.741,174.828,17.365,152.725
C02348=1089.281,-22.575,-54.753,174.829,17.366,152.725
C02349=1089.287,-22.325,-54.766,174.831,17.368,152.725
C02350=1089.293,-22.075,-54.779,174.832,17.370,152.725
C02351=1089.298,-21.825,-54.792,174.835,17.371,152.725
C02352=1089.305,-21.576,-54.805,174.836,17.373,152.725
C02353=1089.310,-21.327,-54.817,174.837,17.374,152.725
C02354=1089.316,-21.077,-54.831,174.839,17.375,152.725
C02355=1089.322,-20.828,-54.843,174.840,17.377,152.725
C02356=1089.328,-20.578,-54.857,174.843,17.379,152.725
C02357=1089.333,-20.328,-54.870,174.844,17.380,152.725
C02358=1089.339,-20.078,-54.882,174.846,17.382,152.725
C02359=1089.346,-19.829,-54.896,174.847,17.384,152.725
C02360=1089.351,-19.579,-54.908,174.849,17.385,152.725
C02361=1089.357,-19.330,-54.922,174.851,17.387,152.725
C02362=1089.363,-19.080,-54.935,174.852,17.388,152.725
C02363=1089.369,-18.830,-54.948,174.854,17.389,152.725
C02364=1089.374,-18.581,-54.960,174.855,17.391,152.725
C02365=1089.381,-18.332,-54.973,174.856,17.393,152.725
C02366=1089.386,-18.082,-54.986,174.858,17.394,152.725
C02367=1089.392,-17.832,-55.000,174.860,17.396,152.725
C02368=1089.398,-17.583,-55.012,174.862,17.397,152.725
C02369=1089.404,-17.333,-55.025,174.863,17.399,152.725
C02370=1089.411,-17.061,-55.040,174.865,17.400,152.725
C02371=1089.417,-16.790,-55.054,174.867,17.402,152.725
C02372=1089.423,-16.518,-55.068,174.868,17.404,152.725
C02373=1089.430,-16.247,-55.083,174.871,17.406,152.725
C02374=1089.435,-15.997,-55.095,174.872,17.407,152.725
C02375=1089.442,-15.748,-55.108,174.873,17.409,152.725
C02376=1089.447,-15.499,-55.122,174.875,17.410,152.725
C02377=1089.453,-15.249,-55.135,174.876,17.411,152.725
C02378=1089.459,-14.999,-55.148,174.879,17.414,152.725
C02379=1089.464,-14.749,-55.161,174.880,17.415,152.725
C02380=1089.471,-14.500,-55.174,174.882,17.416,152.725
C02381=1089.477,-14.251,-55.188,174.883,17.418,152.725
C02382=1089.482,-14.001,-55.201,174.885,17.419,152.724
C02383=1089.488,-13.751,-55.214,174.887,17.421,152.725
C02384=1089.494,-13.502,-55.228,174.888,17.423,152.725
C02385=1089.500,-13.252,-55.240,174.890,17.424,152.725
C02386=1089.506,-13.003,-55.254,174.891,17.425,152.725
C02387=1089.511,-12.752,-55.267,174.893,17.427,152.725
C02388=1089.517,-12.503,-55.280,174.895,17.429,152.725
C02389=1089.523,-12.253,-55.294,174.896,17.431,152.725
C02390=1089.528,-12.004,-55.306,174.898,17.432,152.724
C02391=1089.534,-11.754,-55.320,174.900,17.434,152.724
C02392=1089.540,-11.505,-55.334,174.901,17.436,152.725
C02393=1089.546,-11.256,-55.347,174.903,17.437,152.724
C02394=1089.552,-11.005,-55.360,174.904,17.438,152.724
C02395=1089.558,-10.756,-55.373,174.906,17.440,152.725
C02396=1089.563,-10.506,-55.387,174.908,17.442,152.725
C02397=1089.569,-10.257,-55.400,174.910,17.443,152.724
C02398=1089.575,-10.007,-55.414,174.911,17.445,152.724
C02399=1089.581,-9.758,-55.427,174.912,17.446,152.725
C02400=1089.587,-9.508,-55.440,174.915,17.448,152.724
C02401=1089.592,-9.258,-55.453,174.916,17.449,152.724
C02402=1089.598,-9.009,-55.467,174.918,17.451,152.724
C02403=1089.604,-8.759,-55.480,174.919,17.452,152.724
C02404=1089.610,-8.510,-55.494,174.921,17.454,152.724
C02405=1089.616,-8.261,-55.508,174.923,17.456,152.724
C02406=1089.622,-8.011,-55.520,174.924,17.457,152.724
C02407=1089.627,-7.761,-55.534,174.926,17.459,152.724
C02408=1089.633,-7.512,-55.547,174.927,17.460,152.724
C02409=1089.639,-7.262,-55.561,174.929,17.462,152.724
C02410=1089.646,-7.012,-55.575,174.931,17.463,152.724
C02411=1089.651,-6.762,-55.588,174.932,17.465,152.724
C02412=1089.657,-6.513,-55.601,174.934,17.467,152.724
C02413=1089.662,-6.263,-55.615,174.936,17.468,152.724
C02414=1089.669,-6.014,-55.628,174.938,17.470,152.724
C02415=1089.674,-5.764,-55.642,174.939,17.471,152.724
C02416=1089.680,-5.515,-55.655,174.941,17.472,152.724
C02417=1089.686,-5.266,-55.669,174.943,17.475,152.724
C02418=1089.692,-5.016,-55.683,174.944,17.476,152.724
C02419=1089.697,-4.766,-55.696,174.946,17.477,152.724
C02420=1089.704,-4.516,-55.709,174.947,17.479,152.724
C02421=1089.709,-4.267,-55.723,174.949,17.481,152.724
C02422=1089.716,-4.017,-55.736,174.951,17.482,152.724
C02423=1089.721,-3.768,-55.750,174.952,17.484,152.724
C02424=1089.727,-3.519,-55.764,174.954,17.485,152.724
C02425=1089.733,-3.269,-55.777,174.956,17.487,152.724
C02426=1089.738,-3.019,-55.791,174.958,17.489,152.724
C02427=1089.745,-2.770,-55.805,174.959,17.490,152.724
C02428=1089.750,-2.521,-55.818,174.960,17.492,152.724
C02429=1089.755,-2.271,-55.832,174.963,17.493,152.724
C02430=1089.761,-2.021,-55.846,174.964,17.495,152.724
C02431=1089.768,-1.771,-55.860,174.965,17.497,152.724
C02432=1089.773,-1.522,-55.874,174.967,17.498,152.724
C02433=1089.779,-1.272,-55.888,174.969,17.500,152.724
C02434=1089.785,-1.000,-55.902,174.971,17.501,152.724
C02435=1089.791,-0.726,-55.917,174.973,17.504,152.724
C02436=1089.797,-0.453,-55.933,174.974,17.505,152.724
C02437=1089.804,-0.179,-55.948,174.976,17.507,152.724
C02438=1089.810,0.070,-55.961,174.978,17.508,152.724
C02439=1089.815,0.320,-55.975,174.979,17.510,152.724
C02440=1089.821,0.569,-55.989,174.981,17.512,152.724
C02441=1089.827,0.819,-56.002,174.983,17.514,152.724
C02442=1089.832,1.068,-56.016,174.985,17.515,152.724
C02443=1089.838,1.318,-56.030,174.986,17.516,152.724
C02444=1089.843,1.567,-56.044,174.987,17.518,152.724
C02445=1089.850,1.817,-56.058,174.990,17.520,152.724
C02446=1089.855,2.067,-56.072,174.991,17.521,152.724
C02447=1089.861,2.316,-56.085,174.993,17.523,152.724
C02448=1089.867,2.565,-56.100,174.994,17.524,152.724
C02449=1089.872,2.815,-56.114,174.996,17.526,152.724
C02450=1089.878,3.064,-56.127,174.998,17.528,152.724
C02451=1089.884,3.314,-56.141,174.999,17.529,152.724
C02452=1089.890,3.564,-56.155,175.001,17.531,152.724
C02453=1089.895,3.814,-56.169,175.003,17.532,152.724
C02454=1089.901,4.063,-56.183,175.004,17.534,152.724
C02455=1089.907,4.312,-56.197,175.006,17.536,152.724
C02456=1089.913,4.561,-56.211,175.008,17.537,152.724
C02457=1089.919,4.812,-56.225,175.010,17.539,152.724
C02458=1089.924,5.061,-56.239,175.011,17.540,152.724
C02459=1089.930,5.311,-56.253,175.013,17.542,152.724
C02460=1089.936,5.560,-56.267,175.015,17.544,152.724
C02461=1089.942,5.809,-56.281,175.016,17.545,152.724
C02462=1089.948,6.059,-56.295,175.018,17.546,152.724
C02463=1089.953,6.309,-56.309,175.020,17.548,152.724
C02464=1089.959,6.558,-56.323,175.021,17.550,152.724
C02465=1089.965,6.807,-56.337,175.023,17.551,152.724
C02466=1089.971,7.058,-56.351,175.025,17.553,152.724
C02467=1089.977,7.307,-56.365,175.027,17.555,152.724
C02468=1089.982,7.557,-56.378,175.028,17.556,152.724
C02469=1089.988,7.805,-56.393,175.030,17.558,152.724
C02470=1089.994,8.056,-56.407,175.032,17.560,152.724
C02471=1090.000,8.305,-56.421,175.033,17.561,152.724
C02472=1090.006,8.554,-56.436,175.035,17.562,152.724
C02473=1090.011,8.804,-56.450,175.037,17.565,152.724
C02474=1090.017,9.054,-56.464,175.039,17.566,152.724
C02475=1090.023,9.303,-56.477,175.040,17.567,152.724
C02476=1090.029,9.552,-56.492,175.041,17.569,152.724
C02477=1090.035,9.803,-56.506,175.044,17.570,152.724
C02478=1090.041,10.052,-56.520,175.045,17.572,152.724
C02479=1090.046,10.301,-56.534,175.047,17.574,152.724
C02480=1090.052,10.551,-56.548,175.049,17.575,152.724
C02481=1090.058,10.800,-56.563,175.050,17.577,152.724
C02482=1090.064,11.050,-56.577,175.052,17.578,152.724
C02483=1090.069,11.300,-56.591,175.054,17.580,152.724
C02484=1090.076,11.549,-56.606,175.056,17.582,152.724
C02485=1090.082,11.798,-56.619,175.057,17.583,152.724
C02486=1090.088,12.047,-56.634,175.059,17.584,152.724
C02487=1090.094,12.298,-56.648,175.061,17.586,152.724
C02488=1090.099,12.547,-56.662,175.063,17.588,152.724
C02489=1090.105,12.796,-56.676,175.064,17.589,152.724
C02490=1090.111,13.047,-56.691,175.066,17.591,152.724
C02491=1090.117,13.295,-56.705,175.068,17.592,152.724
C02492=1090.122,13.545,-56.719,175.069,17.594,152.724
C02493=1090.129,13.795,-56.734,175.072,17.596,152.724
C02494=1090.134,14.044,-56.748,175.073,17.597,152.724
C02495=1090.141,14.294,-56.763,175.074,17.599,152.724
C02496=1090.146,14.544,-56.777,175.076,17.600,152.724
C02497=1090.152,14.792,-56.791,175.078,17.602,152.724
C02498=1090.158,15.069,-56.807,175.080,17.604,152.724
C02499=1090.165,15.343,-56.823,175.082,17.605,152.723
C02500=1090.171,15.619,-56.838,175.083,17.607,152.724
C02501=1090.177,15.894,-56.855,175.086,17.609,152.724
C02502=1090.183,16.143,-56.869,175.087,17.610,152.723
C02503=1090.189,16.393,-56.883,175.089,17.612,152.723
C02504=1090.194,16.642,-56.898,175.091,17.614,152.723
C02505=1090.200,16.891,-56.912,175.092,17.615,152.723
C02506=1090.206,17.141,-56.927,175.095,17.617,152.723
C02507=1090.212,17.391,-56.941,175.096,17.619,152.723
C02508=1090.217,17.640,-56.956,175.098,17.620,152.723
C02509=1090.223,17.890,-56.971,175.100,17.622,152.723
C02510=1090.229,18.139,-56.985,175.101,17.623,152.723
C02511=1090.235,18.389,-57.000,175.103,17.624,152.723
C02512=1090.240,18.638,-57.013,175.105,17.627,152.723
C02513=1090.246,18.887,-57.028,175.107,17.628,152.723
C02514=1090.253,19.137,-57.043,175.108,17.629,152.723
C02515=1090.257,19.387,-57.057,175.110,17.631,152.723
C02516=1090.264,19.637,-57.072,175.112,17.633,152.723
C02517=1090.269,19.886,-57.086,175.113,17.634,152.723
C02518=1090.275,20.135,-57.101,175.116,17.636,152.723
C02519=1090.281,20.385,-57.116,175.117,17.637,152.723
C02520=1090.286,20.635,-57.130,175.119,17.639,152.723
C02521=1090.293,20.884,-57.145,175.121,17.641,152.723
C02522=1090.298,21.133,-57.160,175.122,17.642,152.723
C02523=1090.304,21.382,-57.174,175.124,17.644,152.723
C02524=1090.309,21.633,-57.189,175.126,17.645,152.723
C02525=1090.315,21.882,-57.204,175.128,17.647,152.723
C02526=1090.322,22.131,-57.219,175.129,17.648,152.723
C02527=1090.327,22.381,-57.233,175.131,17.650,152.723
C02528=1090.332,22.630,-57.248,175.133,17.652,152.723
C02529=1090.338,22.880,-57.263,175.134,17.653,152.723
C02530=1090.344,23.129,-57.277,175.137,17.655,152.723
C02531=1090.350,23.379,-57.292,175.138,17.656,152.723
C02532=1090.355,23.628,-57.307,175.140,17.658,152.723
C02533=1090.361,23.877,-57.321,175.142,17.660,152.723
C02534=1090.368,24.127,-57.336,175.143,17.661,152.723
C02535=1090.372,24.377,-57.351,175.145,17.662,152.723
C02536=1090.379,24.627,-57.366,175.147,17.664,152.723
C02537=1090.384,24.876,-57.380,175.149,17.666,152.723
C02538=1090.390,25.126,-57.396,175.150,17.667,152.723
C02539=1090.396,25.374,-57.410,175.153,17.669,152.723
C02540=1090.402,25.625,-57.425,175.154,17.670,152.723
C02541=1090.407,25.874,-57.440,175.156,17.672,152.723
C02542=1090.413,26.124,-57.455,175.158,17.674,152.723
C02543=1090.419,26.373,-57.469,175.159,17.675,152.723
C02544=1090.425,26.623,-57.485,175.161,17.676,152.723
C02545=1090.431,26.872,-57.499,175.163,17.678,152.722
C02546=1090.437,27.121,-57.514,175.165,17.680,152.722
C02547=1090.442,27.371,-57.529,175.167,17.682,152.723
C02548=1090.448,27.621,-57.544,175.168,17.683,152.722
C02549=1090.454,27.870,-57.558,175.170,17.684,152.722
C02550=1090.460,28.120,-57.574,175.172,17.686,152.722
C02551=1090.465,28.369,-57.588,175.174,17.688,152.722
C02552=1090.471,28.619,-57.604,175.175,17.689,152.722
C02553=1090.477,28.868,-57.619,175.178,17.691,152.722
C02554=1090.482,29.118,-57.634,175.179,17.692,152.722
C02555=1090.488,29.366,-57.649,175.181,17.694,152.722
C02556=1090.495,29.616,-57.664,175.183,17.696,152.722
C02557=1090.500,29.865,-57.679,175.184,17.697,152.722
C02558=1090.506,30.115,-57.694,175.187,17.699,152.722
C02559=1090.511,30.364,-57.709,175.188,17.700,152.722
C02560=1090.517,30.614,-57.724,175.190,17.702,152.722
C02561=1090.522,30.863,-57.739,175.192,17.703,152.722
C02562=1090.529,31.140,-57.756,175.193,17.705,152.722
C02563=1090.535,31.417,-57.772,175.196,17.707,152.722
C02564=1090.541,31.693,-57.789,175.198,17.709,152.722
C02565=1090.548,31.970,-57.805,175.200,17.710,152.722
C02566=1090.553,32.220,-57.821,175.202,17.712,152.722
C02567=1090.559,32.469,-57.835,175.203,17.713,152.722
C02568=1090.565,32.719,-57.851,175.205,17.714,152.722
C02569=1090.570,32.968,-57.866,175.207,17.717,152.722
C02570=1090.576,33.217,-57.881,175.209,17.718,152.722
C02571=1090.582,33.467,-57.897,175.210,17.719,152.722
C02572=1090.588,33.716,-57.911,175.212,17.721,152.722
C02573=1090.594,33.966,-57.927,175.214,17.722,152.722
C02574=1090.600,34.215,-57.942,175.216,17.725,152.722
C02575=1090.605,34.465,-57.958,175.218,17.726,152.722
C02576=1090.611,34.714,-57.972,175.219,17.727,152.722
C02577=1090.617,34.964,-57.988,175.222,17.729,152.721
C02578=1090.622,35.214,-58.003,175.223,17.730,152.721
C02579=1090.628,35.462,-58.018,175.225,17.732,152.721
C02580=1090.634,35.712,-58.033,175.227,17.733,152.721
C02581=1090.640,35.961,-58.049,175.229,17.735,152.721
C02582=1090.645,36.211,-58.064,175.231,17.736,152.721
C02583=1090.652,36.460,-58.079,175.233,17.738,152.721
C02584=1090.657,36.710,-58.094,175.234,17.739,152.721
C02585=1090.662,36.960,-58.110,175.236,17.741,152.721
C02586=1090.669,37.209,-58.125,175.238,17.742,152.721
C02587=1090.674,37.458,-58.141,175.240,17.744,152.721
C02588=1090.681,37.708,-58.156,175.242,17.746,152.721
C02589=1090.686,37.957,-58.171,175.243,17.747,152.721
C02590=1090.691,38.207,-58.186,175.246,17.749,152.721
C02591=1090.698,38.456,-58.202,175.247,17.750,152.721
C02592=1090.703,38.705,-58.217,175.250,17.752,152.721
C02593=1090.709,38.955,-58.233,175.251,17.754,152.721
C02594=1090.714,39.205,-58.248,175.253,17.755,152.721
C02595=1090.720,39.453,-58.264,175.255,17.757,152.721
C02596=1090.726,39.703,-58.279,175.256,17.758,152.721
C02597=1090.731,39.953,-58.294,175.259,17.759,152.721
C02598=1090.737,40.203,-58.310,175.260,17.761,152.721
C02599=1090.743,40.452,-58.326,175.262,17.762,152.721
C02600=1090.748,40.701,-58.341,175.264,17.764,152.721
C02601=1090.754,40.951,-58.356,175.266,17.765,152.720
C02602=1090.760,41.200,-58.372,175.268,17.768,152.720
C02603=1090.765,41.450,-58.388,175.270,17.769,152.720
C02604=1090.771,41.699,-58.403,175.271,17.770,152.720
C02605=1090.777,41.949,-58.419,175.273,17.772,152.720
C02606=1090.782,42.198,-58.434,175.275,17.773,152.720
C02607=1090.788,42.448,-58.450,175.277,17.775,152.720
C02608=1090.795,42.697,-58.465,175.279,17.776,152.720
C02609=1090.800,42.946,-58.480,175.280,17.778,152.720
C02610=1090.805,43.196,-58.496,175.283,17.779,152.720
C02611=1090.811,43.445,-58.512,175.284,17.781,152.720
C02612=1090.816,43.695,-58.527,175.287,17.783,152.720
C02613=1090.822,43.944,-58.544,175.288,17.784,152.720
C02614=1090.828,44.194,-58.559,175.291,17.786,152.720
C02615=1090.834,44.442,-58.574,175.292,17.787,152.720
C02616=1090.840,44.692,-58.590,175.294,17.788,152.720
C02617=1090.845,44.942,-58.606,175.296,17.790,152.720
C02618=1090.851,45.191,-58.621,175.297,17.792,152.720
C02619=1090.856,45.441,-58.637,175.300,17.793,152.720
C02620=1090.862,45.690,-58.653,175.301,17.795,152.720
C02621=1090.867,45.939,-58.668,175.304,17.797,152.719
C02622=1090.873,46.189,-58.685,175.305,17.798,152.720
C02623=1090.879,46.439,-58.700,175.307,17.799,152.719
C02624=1090.884,46.687,-58.716,175.309,17.801,152.719
C02625=1090.890,46.937,-58.732,175.311,17.802,152.719
C02626=1090.896,47.214,-58.749,175.313,17.804,152.719
C02627=1090.902,47.491,-58.767,175.315,17.806,152.719
C02628=1090.908,47.767,-58.785,175.317,17.807,152.719
C02629=1090.915,48.044,-58.802,175.319,17.809,152.719
C02630=1090.920,48.294,-58.818,175.321,17.810,152.719
C02631=1090.926,48.543,-58.834,175.323,17.813,152.719
C02632=1090.931,48.792,-58.849,175.325,17.814,152.719
C02633=1090.937,49.042,-58.865,175.327,17.815,152.719
C02634=1090.943,49.291,-58.882,175.328,17.817,152.719
C02635=1090.949,49.541,-58.897,175.331,17.819,152.719
C02636=1090.954,49.789,-58.913,175.333,17.820,152.719
C02637=1090.960,50.039,-58.929,175.335,17.822,152.719
C02638=1090.966,50.289,-58.945,175.336,17.823,152.719
C02639=1090.972,50.538,-58.961,175.338,17.824,152.719
C02640=1090.977,50.787,-58.976,175.340,17.826,152.719
C02641=1090.983,51.037,-58.993,175.342,17.827,152.718
C02642=1090.989,51.286,-59.009,175.344,17.829,152.718
C02643=1090.994,51.536,-59.024,175.346,17.830,152.718
C02644=1091.000,51.785,-59.041,175.348,17.832,152.718
C02645=1091.006,52.034,-59.057,175.350,17.834,152.718
C02646=1091.011,52.284,-59.073,175.352,17.835,152.718
C02647=1091.017,52.534,-59.089,175.354,17.836,152.718
C02648=1091.023,52.783,-59.105,175.355,17.837,152.718
C02649=1091.028,53.033,-59.121,175.358,17.839,152.718
C02650=1091.034,53.282,-59.137,175.359,17.841,152.718
C02651=1091.039,53.531,-59.153,175.362,17.842,152.718
C02652=1091.045,53.781,-59.168,175.363,17.844,152.718
C02653=1091.051,54.030,-59.185,175.366,17.845,152.718
C02654=1091.057,54.280,-59.201,175.367,17.846,152.718
C02655=1091.062,54.528,-59.217,175.369,17.849,152.718
C02656=1091.068,54.778,-59.233,175.371,17.850,152.717
C02657=1091.073,55.028,-59.249,175.373,17.851,152.717
C02658=1091.079,55.277,-59.266,175.375,17.852,152.717
C02659=1091.085,55.527,-59.282,175.377,17.854,152.717
C02660=1091.091,55.776,-59.298,175.379,17.856,152.717
C02661=1091.097,56.026,-59.314,175.381,17.857,152.717
C02662=1091.103,56.275,-59.330,175.383,17.858,152.717
C02663=1091.108,56.524,-59.346,175.385,17.859,152.717
C02664=1091.114,56.773,-59.362,175.387,17.862,152.717
C02665=1091.119,57.023,-59.379,175.389,17.863,152.717
C02666=1091.125,57.272,-59.395,175.391,17.864,152.717
C02667=1091.131,57.522,-59.411,175.393,17.865,152.717
C02668=1091.137,57.772,-59.427,175.394,17.867,152.717
C02669=1091.143,58.021,-59.443,175.397,17.869,152.716
C02670=1091.149,58.270,-59.459,175.398,17.870,152.716
C02671=1091.155,58.520,-59.476,175.401,17.871,152.716
C02672=1091.160,58.769,-59.493,175.402,17.872,152.716
C02673=1091.165,59.018,-59.508,175.405,17.874,152.716
C02674=1091.171,59.267,-59.525,175.406,17.876,152.716
C02675=1091.177,59.517,-59.541,175.409,17.877,152.716
C02676=1091.183,59.766,-59.557,175.410,17.878,152.716
C02677=1091.188,60.016,-59.574,175.413,17.880,152.716
C02678=1091.194,60.265,-59.590,175.415,17.881,152.716
C02679=1091.200,60.514,-59.607,175.417,17.883,152.715
C02680=1091.206,60.764,-59.623,175.418,17.884,152.715
C02681=1091.212,61.013,-59.639,175.421,17.886,152.715
C02682=1091.218,61.262,-59.655,175.423,17.887,152.715
C02683=1091.223,61.512,-59.672,175.424,17.888,152.715
C02684=1091.229,61.761,-59.688,175.427,17.890,152.715
C02685=1091.235,62.011,-59.705,175.428,17.891,152.715
C02686=1091.241,62.260,-59.721,175.431,17.892,152.715
C02687=1091.246,62.510,-59.738,175.432,17.893,152.715
C02688=1091.252,62.759,-59.754,175.435,17.895,152.715
C02689=1091.258,63.008,-59.770,175.437,17.896,152.714
C02690=1091.264,63.285,-59.788,175.439,17.898,152.715
C02691=1091.271,63.562,-59.807,175.441,17.900,152.714
C02692=1091.278,63.838,-59.825,175.444,17.902,152.714
C02693=1091.284,64.114,-59.843,175.445,17.903,152.714
C02694=1091.289,64.364,-59.860,175.448,17.904,152.714
C02695=1091.295,64.613,-59.876,175.449,17.905,152.714
C02696=1091.301,64.862,-59.893,175.452,17.907,152.714
C02697=1091.307,65.112,-59.910,175.454,17.908,152.714
C02698=1091.313,65.361,-59.926,175.456,17.910,152.714
C02699=1091.318,65.611,-59.943,175.458,17.911,152.713
C02700=1091.324,65.860,-59.959,175.460,17.913,152.713
C02701=1091.330,66.109,-59.975,175.462,17.914,152.713
C02702=1091.335,66.359,-59.992,175.464,17.916,152.713
C02703=1091.341,66.608,-60.009,175.466,17.917,152.713
C02704=1091.346,66.857,-60.026,175.468,17.918,152.713
C02705=1091.352,67.107,-60.042,175.470,17.919,152.713
C02706=1091.358,67.356,-60.059,175.472,17.921,152.713
C02707=1091.364,67.606,-60.075,175.474,17.922,152.713
C02708=1091.369,67.855,-60.092,175.476,17.924,152.713
C02709=1091.375,68.104,-60.109,175.478,17.925,152.712
C02710=1091.381,68.353,-60.125,175.481,17.927,152.712
C02711=1091.386,68.603,-60.142,175.482,17.928,152.712
C02712=1091.392,68.852,-60.158,175.485,17.929,152.712
C02713=1091.398,69.101,-60.176,175.486,17.931,152.712
C02714=1091.404,69.351,-60.192,175.488,17.932,152.712
C02715=1091.409,69.600,-60.209,175.490,17.934,152.712
C02716=1091.415,69.850,-60.225,175.493,17.935,152.712
C02717=1091.421,70.100,-60.243,175.494,17.936,152.712
C02718=1091.427,70.349,-60.260,175.497,17.938,152.712
C02719=1091.432,70.599,-60.276,175.498,17.939,152.712
C02720=1091.438,70.848,-60.294,175.501,17.941,152.711
C02721=1091.444,71.097,-60.310,175.502,17.942,152.711
C02722=1091.449,71.347,-60.327,175.505,17.943,152.711
C02723=1091.455,71.595,-60.344,175.507,17.944,152.711
C02724=1091.460,71.845,-60.361,175.509,17.946,152.711
C02725=1091.465,72.095,-60.378,175.511,17.947,152.711
C02726=1091.472,72.343,-60.395,175.513,17.949,152.711
C02727=1091.477,72.593,-60.412,175.515,17.950,152.711
C02728=1091.483,72.842,-60.428,175.517,17.951,152.710
C02729=1091.488,73.091,-60.445,175.519,17.953,152.710
C02730=1091.494,73.341,-60.462,175.521,17.954,152.710
C02731=1091.500,73.590,-60.479,175.523,17.955,152.710
C02732=1091.506,73.840,-60.496,175.526,17.957,152.710
C02733=1091.511,74.089,-60.514,175.527,17.958,152.710
C02734=1091.517,74.339,-60.530,175.530,17.960,152.710
C02735=1091.522,74.588,-60.547,175.531,17.961,152.710
C02736=1091.528,74.837,-60.565,175.534,17.962,152.710
C02737=1091.534,75.087,-60.581,175.535,17.963,152.709
C02738=1091.539,75.336,-60.599,175.538,17.965,152.709
C02739=1091.545,75.585,-60.615,175.540,17.966,152.709
C02740=1091.551,75.835,-60.633,175.542,17.968,152.709
C02741=1091.557,76.084,-60.650,175.545,17.969,152.709
C02742=1091.562,76.333,-60.667,175.546,17.970,152.709
C02743=1091.568,76.583,-60.683,175.549,17.972,152.709
C02744=1091.574,76.832,-60.701,175.551,17.973,152.709
C02745=1091.579,77.081,-60.718,175.553,17.974,152.708
C02746=1091.585,77.330,-60.735,175.555,17.975,152.708
C02747=1091.591,77.581,-60.752,175.557,17.977,152.708
C02748=1091.596,77.830,-60.770,175.559,17.978,152.708
C02749=1091.602,78.079,-60.787,175.561,17.980,152.708
C02750=1091.608,78.328,-60.803,175.563,17.981,152.708
C02751=1091.613,78.577,-60.821,175.565,17.982,152.708
C02752=1091.619,78.827,-60.838,175.567,17.984,152.708
C02753=1091.625,79.076,-60.856,175.570,17.985,152.707
C02754=1091.631,79.353,-60.875,175.572,17.986,152.707
C02755=1091.637,79.629,-60.893,175.574,17.987,152.707
C02756=1091.643,79.905,-60.913,175.576,17.989,152.707
C02757=1091.649,80.181,-60.932,175.579,17.991,152.707
C02758=1091.655,80.431,-60.949,175.581,17.992,152.707
C02759=1091.661,80.681,-60.967,175.583,17.993,152.707
C02760=1091.667,80.929,-60.984,175.586,17.995,152.707
C02761=1091.672,81.179,-61.001,175.587,17.996,152.706
C02762=1091.678,81.428,-61.018,175.590,17.998,152.706
C02763=1091.683,81.677,-61.036,175.592,17.998,152.706
C02764=1091.689,81.927,-61.053,175.594,18.000,152.706
C02765=1091.694,82.176,-61.071,175.596,18.001,152.706
C02766=1091.700,82.425,-61.088,175.598,18.003,152.706
C02767=1091.706,82.674,-61.106,175.601,18.004,152.706
C02768=1091.711,82.924,-61.123,175.602,18.005,152.705
C02769=1091.717,83.174,-61.141,175.605,18.007,152.705
C02770=1091.723,83.423,-61.157,175.607,18.008,152.705
C02771=1091.729,83.672,-61.175,175.609,18.009,152.705
C02772=1091.734,83.921,-61.192,175.611,18.010,152.705
C02773=1091.740,84.171,-61.210,175.613,18.012,152.705
C02774=1091.745,84.420,-61.227,175.615,18.013,152.705
C02775=1091.751,84.669,-61.245,175.618,18.014,152.704
C02776=1091.756,84.919,-61.262,175.620,18.016,152.704
C02777=1091.762,85.169,-61.280,175.622,18.017,152.704
C02778=1091.768,85.418,-61.297,175.624,18.019,152.704
C02779=1091.773,85.667,-61.315,175.626,18.020,152.704
C02780=1091.779,85.916,-61.332,175.629,18.021,152.704
C02781=1091.785,86.165,-61.350,175.630,18.022,152.704
C02782=1091.791,86.414,-61.368,175.633,18.024,152.703
C02783=1091.796,86.664,-61.385,175.634,18.025,152.703
C02784=1091.802,86.914,-61.403,175.637,18.026,152.703
C02785=1091.807,87.163,-61.420,175.640,18.027,152.703
C02786=1091.813,87.412,-61.438,175.641,18.028,152.703
C02787=1091.819,87.662,-61.456,175.644,18.030,152.703
C02788=1091.825,87.911,-61.473,175.646,18.031,152.703
C02789=1091.830,88.160,-61.491,175.648,18.032,152.702
C02790=1091.836,88.409,-61.508,175.650,18.033,152.702
C02791=1091.842,88.658,-61.526,175.653,18.035,152.702
C02792=1091.847,88.908,-61.544,175.655,18.036,152.702
C02793=1091.853,89.157,-61.562,175.657,18.037,152.702
C02794=1091.859,89.406,-61.579,175.659,18.038,152.702
C02795=1091.864,89.655,-61.597,175.661,18.039,152.701
C02796=1091.870,89.905,-61.615,175.664,18.041,152.701
C02797=1091.876,90.154,-61.633,175.665,18.042,152.701
C02798=1091.882,90.403,-61.650,175.668,18.043,152.701
C02799=1091.888,90.653,-61.668,175.671,18.044,152.701
C02800=1091.893,90.902,-61.686,175.672,18.046,152.701
C02801=1091.899,91.151,-61.703,175.675,18.047,152.700
C02802=1091.905,91.401,-61.721,175.677,18.048,152.700
C02803=1091.910,91.650,-61.739,175.679,18.049,152.700
C02804=1091.915,91.899,-61.757,175.681,18.051,152.700
C02805=1091.921,92.149,-61.775,175.683,18.052,152.700
C02806=1091.927,92.398,-61.792,175.686,18.053,152.700
C02807=1091.932,92.647,-61.810,175.688,18.054,152.699
C02808=1091.938,92.897,-61.828,175.690,18.056,152.699
C02809=1091.943,93.146,-61.846,175.692,18.057,152.699
C02810=1091.949,93.395,-61.864,175.695,18.058,152.699
C02811=1091.955,93.645,-61.882,175.696,18.059,152.699
C02812=1091.960,93.894,-61.899,175.699,18.060,152.699
C02813=1091.967,94.143,-61.918,175.701,18.062,152.698
C02814=1091.972,94.392,-61.936,175.703,18.063,152.698
C02815=1091.977,94.641,-61.953,175.706,18.064,152.698
C02816=1091.983,94.891,-61.971,175.707,18.065,152.698
C02817=1091.989,95.140,-61.989,175.710,18.067,152.698
C02818=1091.995,95.417,-62.009,175.713,18.068,152.698
C02819=1092.002,95.693,-62.029,175.715,18.069,152.697
C02820=1092.007,95.969,-62.049,175.718,18.071,152.697
C02821=1092.013,96.246,-62.069,175.721,18.072,152.697
C02822=1092.019,96.495,-62.088,175.722,18.073,152.697
C02823=1092.025,96.744,-62.105,175.725,18.074,152.697
C02824=1092.031,96.994,-62.123,175.727,18.075,152.696
C02825=1092.036,97.243,-62.142,175.729,18.077,152.696
C02826=1092.042,97.492,-62.160,175.732,18.078,152.696
C02827=1092.048,97.741,-62.178,175.734,18.079,152.696
C02828=1092.053,97.990,-62.195,175.736,18.080,152.696
C02829=1092.059,98.240,-62.214,175.738,18.081,152.696
C02830=1092.064,98.489,-62.232,175.741,18.083,152.695
C02831=1092.071,98.739,-62.250,175.743,18.084,152.695
C02832=1092.075,98.988,-62.268,175.745,18.085,152.695
C02833=1092.082,99.237,-62.287,175.748,18.086,152.695
C02834=1092.087,99.486,-62.304,175.749,18.087,152.695
C02835=1092.093,99.736,-62.323,175.752,18.089,152.695
C02836=1092.098,99.985,-62.341,175.755,18.090,152.694
C02837=1092.105,100.234,-62.359,175.756,18.091,152.694
C02838=1092.109,100.484,-62.377,175.759,18.092,152.694
C02839=1092.116,100.733,-62.396,175.761,18.093,152.694
C02840=1092.121,100.982,-62.414,175.763,18.094,152.694
C02841=1092.127,101.231,-62.433,175.766,18.095,152.693
C02842=1092.133,101.480,-62.450,175.768,18.097,152.693
C02843=1092.138,101.730,-62.469,175.771,18.098,152.693
C02844=1092.144,101.979,-62.487,175.772,18.099,152.693
C02845=1092.149,102.229,-62.506,175.775,18.100,152.693
C02846=1092.155,102.477,-62.524,175.777,18.102,152.692
C02847=1092.161,102.727,-62.542,175.779,18.102,152.692
C02848=1092.166,102.976,-62.561,175.782,18.104,152.692
C02849=1092.172,103.226,-62.579,175.785,18.105,152.692
C02850=1092.177,103.475,-62.597,175.786,18.106,152.692
C02851=1092.183,103.724,-62.616,175.789,18.107,152.691
C02852=1092.188,103.973,-62.634,175.791,18.108,152.691
C02853=1092.194,104.223,-62.653,175.793,18.109,152.691
C02854=1092.199,104.472,-62.671,175.796,18.111,152.691
C02855=1092.205,104.721,-62.690,175.798,18.112,152.691
C02856=1092.211,104.970,-62.708,175.800,18.113,152.690
C02857=1092.216,105.220,-62.727,175.803,18.114,152.690
C02858=1092.222,105.468,-62.745,175.805,18.115,152.690
C02859=1092.228,105.718,-62.763,175.808,18.116,152.690
C02860=1092.233,105.967,-62.782,175.809,18.117,152.690
C02861=1092.239,106.217,-62.800,175.812,18.118,152.689
C02862=1092.245,106.466,-62.819,175.815,18.119,152.689
C02863=1092.250,106.715,-62.837,175.816,18.121,152.689
C02864=1092.256,106.965,-62.856,175.819,18.122,152.689
C02865=1092.261,107.213,-62.875,175.822,18.123,152.689
C02866=1092.267,107.463,-62.893,175.823,18.124,152.688
C02867=1092.273,107.712,-62.912,175.826,18.125,152.688
C02868=1092.278,107.961,-62.931,175.828,18.126,152.688
C02869=1092.284,108.211,-62.949,175.831,18.127,152.688
C02870=1092.290,108.459,-62.967,175.833,18.128,152.687
C02871=1092.295,108.709,-62.987,175.835,18.129,152.687
C02872=1092.301,108.959,-63.005,175.838,18.131,152.687
C02873=1092.306,109.207,-63.023,175.840,18.132,152.687
C02874=1092.313,109.456,-63.042,175.842,18.132,152.687
C02875=1092.318,109.706,-63.060,175.845,18.134,152.686
C02876=1092.323,109.955,-63.079,175.848,18.135,152.686
C02877=1092.330,110.204,-63.098,175.850,18.136,152.686
C02878=1092.335,110.453,-63.117,175.852,18.137,152.686
C02879=1092.340,110.703,-63.136,175.855,18.139,152.686
C02880=1092.347,110.952,-63.154,175.857,18.139,152.685
C02881=1092.352,111.201,-63.173,175.859,18.140,152.685
C02882=1092.358,111.478,-63.194,175.862,18.141,152.685
C02883=1092.365,111.754,-63.215,175.865,18.143,152.685
C02884=1092.371,112.031,-63.236,175.868,18.144,152.684
C02885=1092.377,112.307,-63.256,175.870,18.145,152.684
C02886=1092.383,112.557,-63.275,175.872,18.146,152.684
C02887=1092.389,112.805,-63.294,175.875,18.147,152.684
C02888=1092.394,113.054,-63.313,175.877,18.148,152.683
C02889=1092.400,113.304,-63.332,175.879,18.149,152.683
C02890=1092.405,113.553,-63.351,175.882,18.151,152.683
C02891=1092.410,113.803,-63.370,175.885,18.152,152.683
C02892=1092.417,114.052,-63.388,175.887,18.152,152.682
C02893=1092.422,114.301,-63.407,175.889,18.153,152.682
C02894=1092.428,114.550,-63.426,175.891,18.155,152.682
C02895=1092.433,114.799,-63.446,175.894,18.156,152.682
C02896=1092.438,115.048,-63.464,175.896,18.157,152.682
C02897=1092.444,115.298,-63.484,175.898,18.157,152.681
C02898=1092.451,115.547,-63.502,175.901,18.159,152.681
C02899=1092.456,115.795,-63.521,175.904,18.160,152.681
C02900=1092.461,116.045,-63.540,175.906,18.161,152.681
C02901=1092.467,116.295,-63.559,175.908,18.162,152.680
C02902=1092.472,116.544,-63.578,175.911,18.164,152.680
C02903=1092.477,116.793,-63.597,175.913,18.165,152.680
C02904=1092.483,117.043,-63.616,175.915,18.165,152.680
C02905=1092.488,117.291,-63.635,175.918,18.166,152.680
C02906=1092.494,117.541,-63.654,175.921,18.168,152.679
C02907=1092.500,117.790,-63.674,175.923,18.168,152.679
C02908=1092.505,118.040,-63.693,175.925,18.170,152.679
C02909=1092.510,118.288,-63.712,175.928,18.171,152.679
C02910=1092.516,118.538,-63.731,175.930,18.172,152.678
C02911=1092.522,118.787,-63.750,175.933,18.173,152.678
C02912=1092.527,119.035,-63.770,175.935,18.174,152.678
C02913=1092.533,119.285,-63.789,175.937,18.174,152.678
C02914=1092.539,119.534,-63.808,175.940,18.176,152.677
C02915=1092.544,119.784,-63.828,175.942,18.177,152.677
C02916=1092.549,120.032,-63.846,175.944,18.178,152.677
C02917=1092.555,120.282,-63.866,175.947,18.179,152.677
C02918=1092.561,120.531,-63.885,175.950,18.180,152.676
C02919=1092.566,120.781,-63.904,175.952,18.181,152.676
C02920=1092.571,121.029,-63.923,175.954,18.182,152.676
C02921=1092.577,121.279,-63.942,175.957,18.183,152.676
C02922=1092.583,121.528,-63.962,175.959,18.184,152.675
C02923=1092.589,121.777,-63.982,175.962,18.185,152.675
C02924=1092.594,122.026,-64.001,175.965,18.186,152.675
C02925=1092.600,122.275,-64.020,175.967,18.187,152.675
C02926=1092.605,122.525,-64.039,175.969,18.188,152.674
C02927=1092.611,122.773,-64.059,175.972,18.189,152.674
C02928=1092.617,123.023,-64.078,175.975,18.190,152.674
C02929=1092.623,123.272,-64.097,175.977,18.191,152.674
C02930=1092.628,123.521,-64.116,175.979,18.192,152.673
C02931=1092.633,123.770,-64.135,175.982,18.193,152.673
C02932=1092.639,124.019,-64.155,175.984,18.194,152.673
C02933=1092.645,124.269,-64.175,175.987,18.195,152.673
C02934=1092.651,124.518,-64.194,175.989,18.196,152.672
C02935=1092.656,124.768,-64.213,175.992,18.197,152.672
C02936=1092.662,125.016,-64.233,175.994,18.198,152.672
C02937=1092.667,125.265,-64.253,175.997,18.199,152.672
C02938=1092.672,125.515,-64.272,176.000,18.200,152.671
C02939=1092.678,125.764,-64.292,176.002,18.200,152.671
C02940=1092.684,126.013,-64.311,176.004,18.202,152.671
C02941=1092.690,126.263,-64.330,176.007,18.203,152.670
C02942=1092.696,126.511,-64.350,176.009,18.203,152.670
C02943=1092.702,126.761,-64.369,176.012,18.205,152.670
C02944=1092.707,127.010,-64.389,176.014,18.206,152.670
C02945=1092.713,127.259,-64.409,176.017,18.207,152.669
C02946=1092.719,127.535,-64.430,176.020,18.208,152.669
C02947=1092.725,127.811,-64.452,176.023,18.209,152.669
C02948=1092.732,128.088,-64.474,176.026,18.210,152.668
C02949=1092.738,128.364,-64.495,176.028,18.211,152.668
C02950=1092.743,128.614,-64.515,176.031,18.211,152.668
C02951=1092.749,128.863,-64.535,176.033,18.212,152.668
C02952=1092.755,129.112,-64.554,176.036,18.213,152.667
C02953=1092.761,129.361,-64.574,176.038,18.214,152.667
C02954=1092.766,129.610,-64.593,176.041,18.215,152.667
C02955=1092.772,129.859,-64.613,176.044,18.216,152.666
C02956=1092.777,130.109,-64.633,176.046,18.217,152.666
C02957=1092.783,130.358,-64.653,176.048,18.218,152.666
C02958=1092.789,130.607,-64.672,176.051,18.219,152.666
C02959=1092.795,130.856,-64.692,176.054,18.220,152.665
C02960=1092.801,131.105,-64.711,176.056,18.220,152.665
C02961=1092.807,131.354,-64.731,176.059,18.221,152.665
C02962=1092.812,131.604,-64.751,176.061,18.222,152.664
C02963=1092.818,131.853,-64.771,176.064,18.223,152.664
C02964=1092.824,132.102,-64.791,176.066,18.224,152.664
C02965=1092.829,132.351,-64.810,176.069,18.225,152.664
C02966=1092.834,132.600,-64.831,176.072,18.226,152.663
C02967=1092.840,132.850,-64.850,176.075,18.227,152.663
C02968=1092.846,133.098,-64.870,176.076,18.228,152.663
C02969=1092.851,133.348,-64.890,176.079,18.228,152.662
C02970=1092.857,133.597,-64.910,176.082,18.229,152.662
C02971=1092.863,133.846,-64.930,176.085,18.231,152.662
C02972=1092.868,134.095,-64.950,176.087,18.231,152.662
C02973=1092.874,134.344,-64.970,176.090,18.232,152.661
C02974=1092.879,134.593,-64.990,176.093,18.233,152.661
C02975=1092.885,134.843,-65.010,176.094,18.234,152.661
C02976=1092.891,135.092,-65.030,176.097,18.235,152.660
C02977=1092.896,135.341,-65.050,176.100,18.236,152.660
C02978=1092.902,135.590,-65.069,176.103,18.237,152.660
C02979=1092.907,135.839,-65.090,176.105,18.237,152.659
C02980=1092.913,136.088,-65.110,176.108,18.238,152.659
C02981=1092.919,136.337,-65.130,176.110,18.240,152.659
C02982=1092.924,136.587,-65.150,176.113,18.240,152.659
C02983=1092.930,136.835,-65.170,176.115,18.241,152.658
C02984=1092.935,137.085,-65.190,176.118,18.242,152.658
C02985=1092.941,137.333,-65.210,176.121,18.243,152.658
C02986=1092.946,137.583,-65.230,176.124,18.244,152.657
C02987=1092.952,137.832,-65.250,176.126,18.244,152.657
C02988=1092.958,138.081,-65.270,176.129,18.245,152.657
C02989=1092.964,138.330,-65.290,176.131,18.246,152.656
C02990=1092.969,138.579,-65.311,176.134,18.247,152.656
C02991=1092.974,138.828,-65.330,176.136,18.248,152.656
C02992=1092.980,139.078,-65.351,176.139,18.249,152.656
C02993=1092.986,139.327,-65.371,176.142,18.250,152.655
C02994=1092.992,139.576,-65.392,176.145,18.250,152.655
C02995=1092.998,139.825,-65.412,176.147,18.252,152.655
C02996=1093.003,140.074,-65.432,176.149,18.252,152.654
C02997=1093.009,140.323,-65.452,176.152,18.253,152.654
C02998=1093.014,140.572,-65.473,176.155,18.254,152.654
C02999=1093.020,140.822,-65.492,176.158,18.255,152.653
C03000=1093.025,141.071,-65.512,176.160,18.255,152.653
C03001=1093.030,141.320,-65.533,176.163,18.257,152.653
C03002=1093.036,141.569,-65.553,176.166,18.257,152.652
C03003=1093.042,141.818,-65.574,176.168,18.258,152.652
C03004=1093.048,142.067,-65.594,176.170,18.259,152.652
C03005=1093.053,142.316,-65.614,176.173,18.260,152.651
C03006=1093.059,142.565,-65.635,176.176,18.261,152.651
C03007=1093.065,142.814,-65.655,176.179,18.261,152.651
C03008=1093.070,143.063,-65.675,176.182,18.263,152.650
C03009=1093.075,143.313,-65.696,176.184,18.263,152.650
C03010=1093.082,143.589,-65.719,176.187,18.264,152.650
C03011=1093.088,143.865,-65.742,176.190,18.265,152.649
C03012=1093.094,144.141,-65.764,176.193,18.266,152.649
C03013=1093.101,144.418,-65.786,176.196,18.267,152.649
C03014=1093.106,144.667,-65.807,176.198,18.268,152.648
C03015=1093.111,144.916,-65.828,176.201,18.268,152.648
C03016=1093.117,145.165,-65.848,176.204,18.269,152.648
C03017=1093.123,145.415,-65.868,176.207,18.270,152.647
C03018=1093.128,145.663,-65.890,176.210,18.271,152.647
C03019=1093.134,145.912,-65.910,176.212,18.271,152.647
C03020=1093.140,146.161,-65.930,176.215,18.273,152.646
C03021=1093.145,146.410,-65.951,176.218,18.273,152.646
C03022=1093.152,146.660,-65.971,176.220,18.274,152.646
C03023=1093.157,146.909,-65.992,176.223,18.274,152.645
C03024=1093.162,147.158,-66.012,176.225,18.276,152.645
C03025=1093.168,147.406,-66.033,176.228,18.276,152.645
C03026=1093.174,147.655,-66.053,176.231,18.277,152.644
C03027=1093.179,147.905,-66.074,176.234,18.278,152.644
C03028=1093.185,148.154,-66.095,176.236,18.278,152.644
C03029=1093.190,148.403,-66.115,176.239,18.279,152.643
C03030=1093.196,148.652,-66.136,176.242,18.280,152.643
C03031=1093.202,148.901,-66.157,176.245,18.281,152.643
C03032=1093.207,149.151,-66.178,176.248,18.282,152.642
C03033=1093.213,149.400,-66.198,176.250,18.283,152.642
C03034=1093.218,149.648,-66.219,176.253,18.283,152.642
C03035=1093.223,149.897,-66.240,176.255,18.284,152.641
C03036=1093.230,150.147,-66.260,176.258,18.285,152.641
C03037=1093.235,150.396,-66.281,176.261,18.286,152.641
C03038=1093.241,150.644,-66.302,176.264,18.287,152.640
C03039=1093.246,150.894,-66.323,176.266,18.287,152.640
C03040=1093.252,151.143,-66.344,176.269,18.288,152.640
C03041=1093.258,151.392,-66.365,176.272,18.289,152.639
C03042=1093.263,151.641,-66.385,176.275,18.290,152.639
C03043=1093.268,151.890,-66.406,176.278,18.291,152.639
C03044=1093.274,152.139,-66.428,176.280,18.291,152.638
C03045=1093.279,152.388,-66.448,176.283,18.292,152.638
C03046=1093.285,152.637,-66.469,176.286,18.293,152.638
C03047=1093.292,152.886,-66.490,176.288,18.294,152.637
C03048=1093.297,153.136,-66.510,176.291,18.295,152.637
C03049=1093.302,153.384,-66.532,176.293,18.295,152.637
C03050=1093.308,153.633,-66.552,176.296,18.296,152.636
C03051=1093.314,153.882,-66.574,176.299,18.297,152.636
C03052=1093.319,154.132,-66.594,176.302,18.297,152.635
C03053=1093.325,154.380,-66.616,176.305,18.298,152.635
C03054=1093.331,154.630,-66.637,176.308,18.299,152.635
C03055=1093.336,154.879,-66.657,176.310,18.299,152.634
C03056=1093.341,155.127,-66.678,176.313,18.300,152.634
C03057=1093.347,155.377,-66.699,176.316,18.301,152.634
C03058=1093.353,155.626,-66.721,176.319,18.302,152.633
C03059=1093.358,155.875,-66.741,176.322,18.302,152.633
C03060=1093.364,156.124,-66.763,176.325,18.304,152.633
C03061=1093.370,156.373,-66.784,176.327,18.304,152.632
C03062=1093.375,156.622,-66.805,176.330,18.304,152.632
C03063=1093.381,156.871,-66.826,176.332,18.306,152.632
C03064=1093.386,157.120,-66.847,176.335,18.306,152.631
C03065=1093.391,157.369,-66.869,176.338,18.307,152.631
C03066=1093.397,157.619,-66.890,176.341,18.308,152.630
C03067=1093.403,157.867,-66.911,176.343,18.308,152.630
C03068=1093.409,158.116,-66.932,176.346,18.309,152.630
C03069=1093.414,158.366,-66.953,176.349,18.310,152.629
C03070=1093.420,158.614,-66.974,176.352,18.311,152.629
C03071=1093.426,158.864,-66.995,176.355,18.311,152.629
C03072=1093.431,159.112,-67.016,176.358,18.312,152.628
C03073=1093.437,159.362,-67.038,176.361,18.313,152.628
C03074=1093.442,159.638,-67.061,176.364,18.314,152.627
C03075=1093.449,159.914,-67.085,176.367,18.314,152.627
C03076=1093.455,160.189,-67.109,176.370,18.315,152.627
C03077=1093.461,160.466,-67.132,176.373,18.316,152.626
C03078=1093.467,160.714,-67.154,176.376,18.316,152.626
C03079=1093.473,160.964,-67.175,176.379,18.317,152.625
C03080=1093.478,161.213,-67.196,176.382,18.318,152.625
C03081=1093.484,161.462,-67.218,176.385,18.319,152.625
C03082=1093.489,161.711,-67.239,176.387,18.319,152.624
C03083=1093.495,161.959,-67.261,176.390,18.320,152.624
C03084=1093.501,162.209,-67.282,176.393,18.321,152.624
C03085=1093.506,162.458,-67.303,176.396,18.322,152.623
C03086=1093.512,162.707,-67.325,176.399,18.322,152.623
C03087=1093.517,162.956,-67.347,176.401,18.323,152.623
C03088=1093.522,163.204,-67.368,176.404,18.324,152.622
C03089=1093.528,163.454,-67.389,176.407,18.325,152.622
C03090=1093.533,163.703,-67.411,176.410,18.325,152.621
C03091=1093.539,163.952,-67.433,176.412,18.326,152.621
C03092=1093.544,164.201,-67.454,176.415,18.327,152.621
C03093=1093.549,164.450,-67.476,176.418,18.327,152.620
C03094=1093.555,164.699,-67.497,176.421,18.328,152.620
C03095=1093.560,164.948,-67.519,176.424,18.329,152.620
C03096=1093.566,165.197,-67.540,176.427,18.330,152.619
C03097=1093.571,165.446,-67.562,176.430,18.331,152.619
C03098=1093.577,165.695,-67.584,176.432,18.331,152.618
C03099=1093.582,165.944,-67.606,176.435,18.332,152.618
C03100=1093.588,166.193,-67.627,176.438,18.332,152.618
C03101=1093.594,166.442,-67.648,176.441,18.333,152.617
C03102=1093.598,166.691,-67.670,176.444,18.334,152.617
C03103=1093.605,166.940,-67.692,176.447,18.335,152.617
C03104=1093.609,167.189,-67.714,176.450,18.335,152.616
C03105=1093.616,167.438,-67.735,176.453,18.336,152.616
C03106=1093.620,167.687,-67.757,176.456,18.337,152.615
C03107=1093.627,167.936,-67.779,176.458,18.337,152.615
C03108=1093.631,168.185,-67.801,176.461,18.338,152.615
C03109=1093.638,168.434,-67.822,176.464,18.339,152.614
C03110=1093.642,168.683,-67.844,176.467,18.340,152.614
C03111=1093.649,168.932,-67.866,176.470,18.340,152.613
C03112=1093.653,169.181,-67.888,176.473,18.341,152.613
C03113=1093.660,169.430,-67.909,176.476,18.342,152.613
C03114=1093.664,169.679,-67.931,176.479,18.342,152.612
C03115=1093.671,169.928,-67.954,176.482,18.343,152.612
C03116=1093.676,170.177,-67.976,176.485,18.344,152.611
C03117=1093.682,170.426,-67.997,176.487,18.344,152.611
C03118=1093.687,170.675,-68.019,176.490,18.345,152.611
C03119=1093.693,170.924,-68.041,176.493,18.345,152.610
C03120=1093.698,171.173,-68.063,176.496,18.346,152.610
C03121=1093.704,171.422,-68.084,176.499,18.347,152.609
C03122=1093.710,171.670,-68.107,176.502,18.347,152.609
C03123=1093.715,171.920,-68.129,176.505,18.348,152.609
C03124=1093.721,172.168,-68.151,176.508,18.349,152.608
C03125=1093.726,172.418,-68.173,176.511,18.349,152.608
C03126=1093.732,172.667,-68.194,176.514,18.350,152.607
C03127=1093.737,172.915,-68.217,176.517,18.351,152.607
C03128=1093.743,173.165,-68.239,176.519,18.351,152.607
C03129=1093.748,173.413,-68.261,176.522,18.352,152.606
C03130=1093.754,173.663,-68.283,176.525,18.352,152.606
C03131=1093.760,173.912,-68.305,176.528,18.353,152.605
C03132=1093.765,174.160,-68.327,176.531,18.354,152.605
C03133=1093.771,174.410,-68.349,176.534,18.354,152.605
C03134=1093.776,174.658,-68.371,176.537,18.355,152.604
C03135=1093.782,174.907,-68.393,176.540,18.356,152.604
C03136=1093.788,175.156,-68.415,176.543,18.357,152.603
C03137=1093.793,175.405,-68.438,176.546,18.357,152.603
C03138=1093.799,175.681,-68.462,176.549,18.357,152.602
C03139=1093.806,175.956,-68.487,176.552,18.358,152.602
C03140=1093.812,176.232,-68.511,176.555,18.359,152.602
C03141=1093.818,176.507,-68.536,176.559,18.360,152.601
C03142=1093.824,176.757,-68.558,176.562,18.360,152.601
C03143=1093.830,177.006,-68.580,176.565,18.361,152.600
C03144=1093.835,177.254,-68.602,176.568,18.362,152.600
C03145=1093.841,177.504,-68.624,176.570,18.362,152.599
C03146=1093.847,177.752,-68.647,176.574,18.362,152.599
C03147=1093.852,178.002,-68.669,176.577,18.363,152.598
C03148=1093.858,178.250,-68.691,176.580,18.363,152.598
C03149=1093.863,178.499,-68.713,176.583,18.364,152.598
C03150=1093.869,178.748,-68.736,176.586,18.365,152.597
C03151=1093.875,178.998,-68.758,176.588,18.366,152.597
C03152=1093.881,179.246,-68.780,176.592,18.366,152.596
C03153=1093.886,179.495,-68.803,176.595,18.367,152.596
C03154=1093.892,179.744,-68.826,176.598,18.367,152.596
C03155=1093.898,179.993,-68.847,176.601,18.368,152.595
C03156=1093.903,180.242,-68.870,176.604,18.368,152.595
C03157=1093.908,180.491,-68.892,176.607,18.369,152.594
C03158=1093.915,180.740,-68.914,176.610,18.370,152.594
C03159=1093.921,180.989,-68.937,176.613,18.370,152.593
C03160=1093.926,181.238,-68.960,176.616,18.370,152.593
C03161=1093.932,181.487,-68.983,176.619,18.371,152.592
C03162=1093.937,181.735,-69.004,176.622,18.372,152.592
C03163=1093.943,181.984,-69.027,176.624,18.372,152.592
C03164=1093.949,182.233,-69.050,176.628,18.372,152.591
C03165=1093.954,182.483,-69.072,176.631,18.373,152.591
C03166=1093.961,182.731,-69.094,176.634,18.374,152.590
C03167=1093.966,182.980,-69.117,176.637,18.374,152.590
C03168=1093.971,183.229,-69.139,176.640,18.375,152.589
C03169=1093.977,183.478,-69.162,176.643,18.375,152.589
C03170=1093.983,183.727,-69.184,176.646,18.376,152.588
C03171=1093.989,183.975,-69.207,176.649,18.376,152.588
C03172=1093.995,184.225,-69.230,176.652,18.377,152.588
C03173=1094.000,184.474,-69.253,176.655,18.377,152.587
C03174=1094.007,184.722,-69.275,176.658,18.378,152.587
C03175=1094.012,184.971,-69.298,176.662,18.378,152.586
C03176=1094.017,185.220,-69.320,176.665,18.379,152.586
C03177=1094.023,185.469,-69.343,176.668,18.380,152.585
C03178=1094.029,185.718,-69.366,176.670,18.380,152.585
C03179=1094.035,185.967,-69.389,176.673,18.381,152.584
C03180=1094.040,186.216,-69.412,176.677,18.381,152.584
C03181=1094.044,186.465,-69.434,176.680,18.382,152.583
C03182=1094.050,186.714,-69.457,176.683,18.383,152.583
C03183=1094.056,186.963,-69.480,176.686,18.383,152.583
C03184=1094.062,187.212,-69.503,176.689,18.384,152.582
C03185=1094.067,187.460,-69.526,176.692,18.384,152.582
C03186=1094.072,187.709,-69.548,176.695,18.385,152.581
C03187=1094.078,187.958,-69.571,176.698,18.386,152.581
C03188=1094.084,188.207,-69.593,176.701,18.386,152.581
C03189=1094.089,188.456,-69.617,176.704,18.387,152.580
C03190=1094.094,188.705,-69.640,176.707,18.387,152.580
C03191=1094.100,188.954,-69.663,176.710,18.388,152.579
C03192=1094.106,189.203,-69.686,176.713,18.389,152.579
C03193=1094.111,189.451,-69.708,176.716,18.389,152.578
C03194=1094.117,189.700,-69.731,176.719,18.390,152.578
C03195=1094.122,189.949,-69.754,176.722,18.390,152.577
C03196=1094.127,190.198,-69.778,176.725,18.391,152.577
C03197=1094.133,190.447,-69.801,176.729,18.391,152.576
C03198=1094.139,190.696,-69.824,176.732,18.392,152.576
C03199=1094.144,190.945,-69.847,176.735,18.393,152.576
C03200=1094.150,191.194,-69.870,176.738,18.393,152.575
C03201=1094.155,191.443,-69.893,176.741,18.394,152.575
C03202=1094.162,191.718,-69.918,176.744,18.394,152.574
C03203=1094.168,191.993,-69.944,176.748,18.395,152.574
C03204=1094.174,192.269,-69.969,176.751,18.396,152.573
C03205=1094.180,192.544,-69.995,176.754,18.396,152.573
C03206=1094.186,192.793,-70.018,176.757,18.396,152.572
C03207=1094.192,193.042,-70.041,176.760,18.397,152.572
C03208=1094.197,193.291,-70.065,176.763,18.398,152.571
C03209=1094.202,193.540,-70.088,176.767,18.398,152.571
C03210=1094.207,193.788,-70.110,176.770,18.399,152.571
C03211=1094.213,194.036,-70.134,176.773,18.399,152.570
C03212=1094.218,194.285,-70.158,176.777,18.400,152.570
C03213=1094.224,194.534,-70.181,176.780,18.401,152.569
C03214=1094.230,194.783,-70.203,176.783,18.401,152.569
C03215=1094.236,195.032,-70.226,176.786,18.402,152.568
C03216=1094.241,195.281,-70.251,176.789,18.402,152.568
C03217=1094.247,195.530,-70.274,176.792,18.403,152.567
C03218=1094.253,195.779,-70.297,176.795,18.404,152.567
C03219=1094.259,196.028,-70.320,176.798,18.404,152.566
C03220=1094.264,196.277,-70.343,176.801,18.405,152.566
C03221=1094.270,196.526,-70.367,176.805,18.405,152.565
C03222=1094.276,196.774,-70.390,176.808,18.406,152.565
C03223=1094.281,197.024,-70.414,176.811,18.406,152.564
C03224=1094.287,197.272,-70.437,176.814,18.407,152.564
C03225=1094.292,197.521,-70.460,176.817,18.407,152.563
C03226=1094.297,197.770,-70.484,176.820,18.408,152.563
C03227=1094.303,198.018,-70.507,176.823,18.408,152.563
C03228=1094.309,198.267,-70.530,176.826,18.409,152.562
C03229=1094.314,198.516,-70.554,176.829,18.409,152.562
C03230=1094.320,198.765,-70.578,176.832,18.410,152.561
C03231=1094.326,199.014,-70.600,176.836,18.410,152.561
C03232=1094.331,199.262,-70.625,176.839,18.410,152.560
C03233=1094.337,199.512,-70.648,176.842,18.411,152.560
C03234=1094.343,199.761,-70.671,176.845,18.411,152.559
C03235=1094.348,200.009,-70.695,176.848,18.412,152.559
C03236=1094.354,200.258,-70.718,176.852,18.413,152.558
C03237=1094.360,200.506,-70.742,176.855,18.413,152.558
C03238=1094.365,200.756,-70.765,176.858,18.413,152.557
C03239=1094.371,201.004,-70.789,176.861,18.414,152.557
C03240=1094.378,201.254,-70.812,176.865,18.414,152.556
C03241=1094.383,201.502,-70.837,176.868,18.415,152.556
C03242=1094.389,201.751,-70.860,176.871,18.415,152.555
C03243=1094.394,202.000,-70.884,176.874,18.416,152.555
C03244=1094.400,202.249,-70.907,176.877,18.416,152.554
C03245=1094.406,202.497,-70.930,176.880,18.417,152.554
C03246=1094.411,202.747,-70.954,176.883,18.417,152.553
C03247=1094.417,202.995,-70.978,176.887,18.418,152.553
C03248=1094.423,203.244,-71.002,176.890,18.418,152.553
C03249=1094.428,203.493,-71.026,176.893,18.419,152.552
C03250=1094.434,203.741,-71.049,176.897,18.420,152.552
C03251=1094.439,203.990,-71.073,176.900,18.420,152.551
C03252=1094.445,204.239,-71.097,176.903,18.421,152.551
C03253=1094.451,204.488,-71.121,176.906,18.421,152.550
C03254=1094.456,204.737,-71.145,176.909,18.422,152.550
C03255=1094.462,204.985,-71.168,176.912,18.422,152.549
C03256=1094.467,205.234,-71.193,176.915,18.423,152.549
C03257=1094.473,205.483,-71.216,176.919,18.423,152.548
C03258=1094.479,205.732,-71.240,176.922,18.424,152.548
C03259=1094.484,205.981,-71.265,176.925,18.424,152.547
C03260=1094.490,206.230,-71.288,176.928,18.424,152.547
C03261=1094.495,206.478,-71.312,176.932,18.426,152.546
C03262=1094.500,206.727,-71.336,176.935,18.426,152.546
C03263=1094.507,206.976,-71.360,176.938,18.427,152.545
C03264=1094.512,207.225,-71.384,176.941,18.427,152.545
C03265=1094.517,207.474,-71.408,176.944,18.428,152.544
C03266=1094.540,208.489,-71.506,176.999,18.451,152.539
C03267=1094.549,208.863,-71.542,177.004,18.453,152.539
C03268=1094.557,209.239,-71.579,177.009,18.456,152.539
C03269=1094.566,209.613,-71.615,177.014,18.458,152.538
C03270=1094.574,209.987,-71.652,177.018,18.460,152.538
C03271=1094.580,210.237,-71.677,177.021,18.461,152.538
C03272=1094.585,210.485,-71.701,177.024,18.463,152.537
C03273=1094.591,210.735,-71.726,177.027,18.464,152.537
C03274=1094.596,210.983,-71.750,177.030,18.465,152.537
C03275=1094.602,211.232,-71.774,177.033,18.467,152.536
C03276=1094.608,211.480,-71.800,177.036,18.468,152.536
C03277=1094.614,211.729,-71.823,177.040,18.470,152.536
C03278=1094.619,211.977,-71.848,177.042,18.471,152.536
C03279=1094.625,212.227,-71.872,177.045,18.472,152.535
C03280=1094.631,212.475,-71.896,177.049,18.474,152.535
C03281=1094.636,212.724,-71.921,177.051,18.475,152.535
C03282=1094.642,212.972,-71.946,177.055,18.477,152.535
C03283=1094.647,213.221,-71.970,177.058,18.478,152.534
C03284=1094.653,213.470,-71.995,177.060,18.479,152.534
C03285=1094.659,213.719,-72.019,177.064,18.481,152.534
C03286=1094.665,213.967,-72.044,177.067,18.482,152.534
C03287=1094.669,214.216,-72.069,177.070,18.484,152.533
C03288=1094.675,214.465,-72.094,177.073,18.485,152.533
C03289=1094.680,214.714,-72.118,177.077,18.487,152.533
C03290=1094.686,214.962,-72.143,177.079,18.488,152.533
C03291=1094.692,215.212,-72.168,177.082,18.489,152.532
C03292=1094.697,215.460,-72.192,177.086,18.491,152.532
C03293=1094.703,215.709,-72.217,177.088,18.492,152.532
C03294=1094.709,215.957,-72.242,177.092,18.494,152.532
C03295=1094.714,216.206,-72.266,177.095,18.495,152.531
C03296=1094.720,216.455,-72.292,177.098,18.497,152.531
C03297=1094.725,216.704,-72.316,177.101,18.498,152.531
C03298=1094.731,216.952,-72.341,177.104,18.499,152.531
C03299=1094.736,217.201,-72.366,177.107,18.501,152.530
C03300=1094.742,217.450,-72.390,177.110,18.502,152.530
C03301=1094.748,217.698,-72.415,177.113,18.504,152.530
C03302=1094.753,217.948,-72.441,177.116,18.505,152.530
C03303=1094.759,218.196,-72.465,177.120,18.507,152.529
C03304=1094.765,218.445,-72.490,177.122,18.508,152.529
C03305=1094.770,218.693,-72.515,177.126,18.510,152.529
C03306=1094.776,218.942,-72.540,177.129,18.511,152.529
C03307=1094.782,219.190,-72.565,177.132,18.512,152.528
C03308=1094.787,219.440,-72.590,177.135,18.514,152.528
C03309=1094.793,219.688,-72.615,177.138,18.515,152.528
C03310=1094.798,219.937,-72.639,177.141,18.516,152.527
C03311=1094.805,220.186,-72.665,177.144,18.518,152.527
C03312=1094.809,220.435,-72.690,177.148,18.519,152.527
C03313=1094.815,220.683,-72.715,177.150,18.521,152.527
C03314=1094.821,220.931,-72.740,177.154,18.522,152.526
C03315=1094.827,221.180,-72.765,177.157,18.524,152.526
C03316=1094.833,221.429,-72.790,177.160,18.525,152.526
C03317=1094.838,221.677,-72.816,177.163,18.527,152.526
C03318=1094.844,221.927,-72.840,177.166,18.528,152.525
C03319=1094.852,222.305,-72.879,177.171,18.530,152.525
C03320=1094.861,222.684,-72.917,177.175,18.532,152.525
C03321=1094.869,223.061,-72.955,177.180,18.534,152.524
C03322=1094.878,223.441,-72.993,177.185,18.537,152.524
C03323=1094.883,223.690,-73.019,177.188,18.538,152.524
C03324=1094.889,223.938,-73.044,177.192,18.540,152.523
C03325=1094.894,224.187,-73.070,177.194,18.541,152.523
C03326=1094.900,224.435,-73.094,177.198,18.543,152.523
C03327=1094.906,224.684,-73.120,177.201,18.544,152.523
C03328=1094.911,224.933,-73.146,177.204,18.546,152.522
C03329=1094.917,225.181,-73.171,177.207,18.547,152.522
C03330=1094.922,225.430,-73.197,177.210,18.549,152.522
C03331=1094.928,225.679,-73.221,177.213,18.550,152.522
C03332=1094.933,225.927,-73.247,177.217,18.552,152.521
C03333=1094.939,226.176,-73.272,177.219,18.553,152.521
C03334=1094.945,226.425,-73.298,177.223,18.555,152.521
C03335=1094.950,226.673,-73.323,177.226,18.556,152.521
C03336=1094.956,226.922,-73.349,177.229,18.558,152.520
C03337=1094.962,227.171,-73.374,177.232,18.559,152.520
C03338=1094.967,227.419,-73.400,177.235,18.561,152.520
C03339=1094.973,227.668,-73.425,177.238,18.562,152.520
C03340=1094.978,227.917,-73.450,177.242,18.564,152.519
C03341=1094.984,228.165,-73.475,177.244,18.565,152.519
C03342=1094.989,228.414,-73.501,177.248,18.567,152.519
C03343=1094.996,228.663,-73.527,177.251,18.568,152.519
C03344=1095.001,228.912,-73.553,177.254,18.570,152.518
C03345=1095.007,229.160,-73.577,177.257,18.571,152.518
C03346=1095.012,229.409,-73.603,177.260,18.573,152.518
C03347=1095.018,229.657,-73.629,177.263,18.574,152.518
C03348=1095.024,229.906,-73.655,177.267,18.576,152.517
C03349=1095.030,230.154,-73.680,177.269,18.577,152.517
C03350=1095.035,230.403,-73.706,177.273,18.579,152.517
C03351=1095.041,230.652,-73.732,177.276,18.580,152.517
C03352=1095.047,230.900,-73.758,177.279,18.582,152.516
C03353=1095.052,231.149,-73.783,177.282,18.583,152.516
C03354=1095.057,231.398,-73.809,177.286,18.585,152.516
C03355=1095.063,231.646,-73.834,177.288,18.586,152.516
C03356=1095.069,231.895,-73.860,177.292,18.588,152.516
C03357=1095.074,232.143,-73.887,177.294,18.589,152.515
C03358=1095.080,232.392,-73.912,177.298,18.591,152.515
C03359=1095.086,232.641,-73.938,177.301,18.592,152.515
C03360=1095.091,232.890,-73.964,177.304,18.594,152.515
C03361=1095.097,233.138,-73.990,177.308,18.596,152.514
C03362=1095.102,233.386,-74.015,177.310,18.597,152.514
C03363=1095.108,233.635,-74.041,177.314,18.599,152.514
C03364=1095.113,233.884,-74.067,177.317,18.600,152.514
C03365=1095.119,234.133,-74.093,177.320,18.602,152.513
C03366=1095.125,234.381,-74.119,177.323,18.603,152.513
C03367=1095.130,234.629,-74.145,177.326,18.605,152.513
C03368=1095.136,234.878,-74.171,177.329,18.606,152.513
C03369=1095.141,235.127,-74.197,177.333,18.608,152.512
C03370=1095.147,235.375,-74.223,177.335,18.609,152.512
C03371=1095.155,235.745,-74.262,177.341,18.612,152.512
C03372=1095.164,236.115,-74.300,177.345,18.614,152.512
C03373=1095.172,236.485,-74.339,177.349,18.616,152.511
C03374=1095.180,236.855,-74.379,177.355,18.619,152.511
C03375=1095.186,237.104,-74.405,177.357,18.620,152.511
C03376=1095.192,237.353,-74.430,177.361,18.622,152.510
C03377=1095.197,237.600,-74.456,177.363,18.624,152.510
C03378=1095.203,237.849,-74.482,177.367,18.625,152.510
C03379=1095.208,238.098,-74.509,177.371,18.627,152.510
C03380=1095.214,238.347,-74.535,177.373,18.628,152.510
C03381=1095.220,238.595,-74.561,177.377,18.630,152.509
C03382=1095.225,238.844,-74.587,177.380,18.631,152.509
C03383=1095.231,239.092,-74.614,177.383,18.633,152.509
C03384=1095.236,239.341,-74.640,177.386,18.634,152.509
C03385=1095.242,239.590,-74.667,177.389,18.636,152.508
C03386=1095.248,239.839,-74.693,177.393,18.638,152.508
C03387=1095.253,240.087,-74.719,177.396,18.639,152.508
C03388=1095.260,240.335,-74.745,177.399,18.641,152.508
C03389=1095.265,240.584,-74.771,177.402,18.642,152.507
C03390=1095.271,240.832,-74.798,177.405,18.644,152.507
C03391=1095.276,241.081,-74.823,177.409,18.646,152.507
C03392=1095.282,241.329,-74.850,177.411,18.647,152.507
C03393=1095.287,241.577,-74.877,177.415,18.649,152.507
C03394=1095.293,241.826,-74.903,177.418,18.650,152.506
C03395=1095.299,242.075,-74.929,177.421,18.652,152.506
C03396=1095.304,242.323,-74.957,177.424,18.653,152.506
C03397=1095.309,242.572,-74.982,177.427,18.655,152.506
C03398=1095.315,242.821,-75.009,177.431,18.657,152.505
C03399=1095.321,243.069,-75.036,177.433,18.658,152.505
C03400=1095.327,243.317,-75.062,177.437,18.660,152.505
C03401=1095.332,243.566,-75.088,177.441,18.662,152.505
C03402=1095.338,243.815,-75.115,177.443,18.663,152.504
C03403=1095.344,244.063,-75.142,177.447,18.665,152.504
C03404=1095.349,244.312,-75.168,177.449,18.667,152.504
C03405=1095.354,244.560,-75.196,177.453,18.668,152.504
C03406=1095.360,244.809,-75.221,177.456,18.670,152.504
C03407=1095.366,245.058,-75.248,177.459,18.671,152.503
C03408=1095.371,245.306,-75.275,177.463,18.673,152.503
C03409=1095.377,245.554,-75.301,177.465,18.675,152.503
C03410=1095.382,245.803,-75.329,177.469,18.677,152.503
C03411=1095.388,246.051,-75.355,177.472,18.678,152.503
C03412=1095.394,246.300,-75.382,177.475,18.680,152.502
C03413=1095.400,246.549,-75.408,177.478,18.681,152.502
C03414=1095.406,246.798,-75.435,177.482,18.684,152.502
C03415=1095.411,247.046,-75.462,177.484,18.685,152.502
C03416=1095.416,247.295,-75.489,177.488,18.686,152.501
C03417=1095.422,247.543,-75.515,177.491,18.688,152.501
C03418=1095.427,247.792,-75.543,177.494,18.689,152.501
C03419=1095.433,248.040,-75.569,177.498,18.692,152.501
C03420=1095.439,248.288,-75.596,177.500,18.693,152.501
C03421=1095.444,248.537,-75.623,177.504,18.695,152.500
C03422=1095.450,248.785,-75.650,177.507,18.697,152.500
C03423=1095.458,249.149,-75.689,177.511,18.699,152.500
C03424=1095.466,249.511,-75.729,177.516,18.702,152.500
C03425=1095.474,249.874,-75.768,177.521,18.704,152.499
C03426=1095.482,250.238,-75.808,177.526,18.706,152.499
C03427=1095.487,250.486,-75.835,177.529,18.709,152.499
C03428=1095.493,250.734,-75.862,177.532,18.710,152.499
C03429=1095.498,250.983,-75.889,177.535,18.712,152.498
C03430=1095.504,251.231,-75.916,177.538,18.714,152.498
C03431=1095.509,251.480,-75.943,177.541,18.715,152.498
C03432=1095.515,251.728,-75.970,177.545,18.717,152.498
C03433=1095.521,251.977,-75.998,177.548,18.719,152.498
C03434=1095.527,252.226,-76.024,177.551,18.720,152.498
C03435=1095.532,252.474,-76.052,177.554,18.722,152.497
C03436=1095.537,252.723,-76.078,177.558,18.724,152.497
C03437=1095.543,252.971,-76.106,177.560,18.725,152.497
C03438=1095.549,253.219,-76.133,177.564,18.727,152.497
C03439=1095.554,253.468,-76.160,177.567,18.729,152.497
C03440=1095.560,253.716,-76.188,177.570,18.731,152.496
C03441=1095.565,253.965,-76.215,177.573,18.732,152.496
C03442=1095.571,254.213,-76.242,177.577,18.734,152.496
C03443=1095.576,254.462,-76.269,177.580,18.735,152.496
C03444=1095.582,254.710,-76.296,177.583,18.738,152.496
C03445=1095.588,254.959,-76.324,177.586,18.739,152.495
C03446=1095.594,255.207,-76.351,177.590,18.741,152.495
C03447=1095.599,255.455,-76.379,177.592,18.743,152.495
C03448=1095.605,255.704,-76.405,177.596,18.745,152.495
C03449=1095.611,255.953,-76.434,177.600,18.746,152.495
C03450=1095.616,256.201,-76.460,177.602,18.748,152.494
C03451=1095.622,256.449,-76.488,177.606,18.750,152.494
C03452=1095.627,256.698,-76.515,177.609,18.752,152.494
C03453=1095.633,256.946,-76.543,177.612,18.753,152.494
C03454=1095.639,257.195,-76.570,177.615,18.755,152.494
C03455=1095.645,257.442,-76.598,177.619,18.757,152.493
C03456=1095.650,257.692,-76.625,177.621,18.758,152.493
C03457=1095.656,257.940,-76.653,177.625,18.760,152.493
C03458=1095.661,258.188,-76.680,177.628,18.762,152.493
C03459=1095.667,258.436,-76.708,177.632,18.764,152.493
C03460=1095.673,258.685,-76.735,177.634,18.765,152.492
C03461=1095.678,258.933,-76.763,177.638,18.767,152.492
C03462=1095.683,259.182,-76.790,177.641,18.769,152.492
C03463=1095.690,259.430,-76.818,177.644,18.770,152.492
C03464=1095.695,259.679,-76.846,177.648,18.772,152.492
C03465=1095.700,259.927,-76.873,177.651,18.774,152.491
C03466=1095.707,260.176,-76.901,177.654,18.776,152.491
C03467=1095.713,260.424,-76.929,177.657,18.777,152.491
C03468=1095.719,260.673,-76.956,177.660,18.780,152.491
C03469=1095.724,260.921,-76.984,177.664,18.781,152.491
C03470=1095.730,261.169,-77.012,177.667,18.783,152.490
C03471=1095.736,261.418,-77.039,177.670,18.785,152.490
C03472=1095.741,261.666,-77.067,177.673,18.787,152.490
C03473=1095.747,261.915,-77.095,177.677,18.788,152.490
C03474=1095.753,262.163,-77.123,177.680,18.790,152.490
C03475=1095.761,262.523,-77.163,177.685,18.792,152.489
C03476=1095.769,262.883,-77.203,177.689,18.795,152.489
C03477=1095.778,263.243,-77.243,177.694,18.797,152.489
C03478=1095.786,263.603,-77.283,177.699,18.800,152.489
C03479=1095.792,263.852,-77.311,177.702,18.802,152.488
C03480=1095.798,264.100,-77.339,177.705,18.803,152.488
C03481=1095.804,264.349,-77.367,177.708,18.805,152.488
C03482=1095.809,264.597,-77.395,177.712,18.808,152.488
C03483=1095.815,264.845,-77.424,177.715,18.809,152.488
C03484=1095.820,265.094,-77.452,177.718,18.811,152.488
C03485=1095.826,265.341,-77.479,177.721,18.813,152.487
C03486=1095.832,265.591,-77.507,177.725,18.815,152.487
C03487=1095.837,265.839,-77.535,177.728,18.817,152.487
C03488=1095.843,266.087,-77.563,177.731,18.818,152.487
C03489=1095.848,266.335,-77.591,177.734,18.820,152.487
C03490=1095.854,266.584,-77.619,177.738,18.822,152.486
C03491=1095.860,266.832,-77.647,177.741,18.824,152.486
C03492=1095.865,267.080,-77.675,177.744,18.825,152.486
C03493=1095.871,267.329,-77.703,177.747,18.828,152.486
C03494=1095.876,267.577,-77.731,177.750,18.829,152.486
C03495=1095.883,267.825,-77.760,177.754,18.832,152.486
C03496=1095.888,268.073,-77.788,177.756,18.833,152.485
C03497=1095.894,268.322,-77.817,177.760,18.835,152.485
C03498=1095.899,268.570,-77.845,177.763,18.837,152.485
C03499=1095.905,268.819,-77.873,177.767,18.839,152.485
C03500=1095.911,269.067,-77.901,177.770,18.841,152.485
C03501=1095.916,269.316,-77.929,177.773,18.843,152.485
C03502=1095.922,269.564,-77.957,177.776,18.844,152.484
C03503=1095.928,269.812,-77.986,177.779,18.847,152.484
C03504=1095.933,270.060,-78.014,177.783,18.848,152.484
C03505=1095.939,270.309,-78.043,177.785,18.850,152.484
C03506=1095.944,270.557,-78.071,177.789,18.852,152.484
C03507=1095.950,270.806,-78.100,177.792,18.854,152.484
C03508=1095.956,271.053,-78.128,177.796,18.856,152.484
C03509=1095.962,271.302,-78.157,177.799,18.858,152.483
C03510=1095.967,271.550,-78.184,177.802,18.859,152.483
C03511=1095.973,271.799,-78.213,177.805,18.862,152.483
C03512=1095.978,272.047,-78.242,177.809,18.863,152.483
C03513=1095.984,272.295,-78.270,177.812,18.866,152.483
C03514=1095.990,272.544,-78.299,177.815,18.868,152.483
C03515=1095.995,272.791,-78.327,177.818,18.869,152.482
C03516=1096.001,273.040,-78.356,177.821,18.871,152.482
C03517=1096.007,273.288,-78.384,177.825,18.873,152.482
C03518=1096.012,273.537,-78.413,177.828,18.875,152.482
C03519=1096.018,273.785,-78.442,177.832,18.877,152.482
C03520=1096.023,274.033,-78.470,177.834,18.879,152.482
C03521=1096.030,274.282,-78.499,177.837,18.881,152.482
C03522=1096.034,274.530,-78.527,177.841,18.883,152.481
C03523=1096.040,274.778,-78.556,177.844,18.885,152.481
C03524=1096.046,275.027,-78.585,177.847,18.887,152.481
C03525=1096.051,275.275,-78.614,177.851,18.889,152.481
C03526=1096.057,275.523,-78.642,177.853,18.891,152.481
C03527=1096.065,275.886,-78.684,177.859,18.894,152.481
C03528=1096.074,276.249,-78.726,177.864,18.897,152.481
C03529=1096.082,276.612,-78.768,177.868,18.899,152.480
C03530=1096.090,276.974,-78.810,177.873,18.903,152.480
C03531=1096.096,277.223,-78.839,177.876,18.905,152.480
C03532=1096.102,277.471,-78.868,177.879,18.906,152.480
C03533=1096.107,277.719,-78.897,177.882,18.908,152.480
C03534=1096.113,277.968,-78.925,177.885,18.911,152.480
C03535=1096.119,278.216,-78.955,177.889,18.912,152.479
C03536=1096.124,278.464,-78.984,177.892,18.915,152.479
C03537=1096.130,278.712,-79.012,177.896,18.917,152.479
C03538=1096.136,278.961,-79.042,177.898,18.918,152.479
C03539=1096.141,279.208,-79.070,177.902,18.920,152.479
C03540=1096.146,279.457,-79.099,177.905,18.923,152.479
C03541=1096.153,279.705,-79.128,177.908,18.925,152.479
C03542=1096.158,279.953,-79.158,177.912,18.927,152.479
C03543=1096.164,280.201,-79.187,177.915,18.929,152.478
C03544=1096.169,280.450,-79.215,177.918,18.931,152.478
C03545=1096.175,280.698,-79.245,177.921,18.932,152.478
C03546=1096.181,280.946,-79.273,177.924,18.934,152.478
C03547=1096.186,281.194,-79.303,177.928,18.937,152.478
C03548=1096.192,281.443,-79.331,177.931,18.939,152.478
C03549=1096.198,281.691,-79.361,177.934,18.941,152.478
C03550=1096.203,281.939,-79.390,177.938,18.943,152.478
C03551=1096.209,282.187,-79.419,177.941,18.945,152.478
C03552=1096.215,282.436,-79.449,177.943,18.947,152.477
C03553=1096.220,282.683,-79.477,177.947,18.949,152.477
C03554=1096.226,282.932,-79.507,177.950,18.951,152.477
C03555=1096.231,283.180,-79.537,177.953,18.954,152.477
C03556=1096.238,283.428,-79.566,177.957,18.955,152.477
C03557=1096.242,283.677,-79.594,177.960,18.958,152.477
C03558=1096.248,283.925,-79.624,177.963,18.960,152.477
C03559=1096.254,284.173,-79.653,177.967,18.962,152.477
C03560=1096.259,284.422,-79.683,177.969,18.964,152.477
C03561=1096.265,284.670,-79.712,177.972,18.966,152.477
C03562=1096.271,284.917,-79.741,177.976,18.968,152.476
C03563=1096.276,285.166,-79.771,177.979,18.970,152.476
C03564=1096.282,285.414,-79.800,177.983,18.972,152.476
C03565=1096.288,285.663,-79.829,177.986,18.974,152.476
C03566=1096.294,285.910,-79.860,177.989,18.977,152.476
C03567=1096.299,286.158,-79.889,177.992,18.979,152.476
C03568=1096.305,286.406,-79.918,177.996,18.981,152.476
C03569=1096.310,286.655,-79.947,177.998,18.983,152.476
C03570=1096.316,286.903,-79.977,178.001,18.985,152.476
C03571=1096.322,287.151,-80.006,178.005,18.987,152.476
C03572=1096.328,287.400,-80.036,178.008,18.989,152.475
C03573=1096.333,287.648,-80.065,178.012,18.991,152.475
C03574=1096.338,287.895,-80.095,178.015,18.994,152.475
C03575=1096.345,288.143,-80.124,178.018,18.996,152.475
C03576=1096.350,288.392,-80.154,178.021,18.998,152.475
C03577=1096.356,288.640,-80.184,178.025,19.000,152.475
C03578=1096.361,288.888,-80.214,178.028,19.003,152.475
C03579=1096.370,289.260,-80.257,178.033,19.006,152.475
C03580=1096.379,289.633,-80.302,178.037,19.009,152.475
C03581=1096.387,290.005,-80.347,178.042,19.012,152.475
C03582=1096.395,290.377,-80.392,178.047,19.015,152.474
C03583=1096.401,290.625,-80.421,178.050,19.018,152.474
C03584=1096.407,290.873,-80.451,178.054,19.020,152.474
C03585=1096.413,291.121,-80.481,178.057,19.022,152.474
C03586=1096.418,291.369,-80.511,178.060,19.024,152.474
C03587=1096.424,291.618,-80.541,178.063,19.027,152.474
C03588=1096.430,291.866,-80.571,178.067,19.029,152.474
C03589=1096.435,292.114,-80.601,178.070,19.031,152.474
C03590=1096.441,292.362,-80.630,178.073,19.033,152.474
C03591=1096.446,292.610,-80.661,178.077,19.035,152.474
C03592=1096.452,292.859,-80.690,178.080,19.038,152.474
C03593=1096.458,293.107,-80.721,178.083,19.040,152.474
C03594=1096.463,293.355,-80.750,178.086,19.042,152.473
C03595=1096.469,293.603,-80.781,178.090,19.044,152.473
C03596=1096.475,293.851,-80.810,178.092,19.047,152.473
C03597=1096.480,294.099,-80.841,178.095,19.049,152.473
C03598=1096.486,294.347,-80.870,178.099,19.051,152.473
C03599=1096.492,294.595,-80.901,178.102,19.053,152.473
C03600=1096.498,294.843,-80.931,178.105,19.056,152.473
C03601=1096.503,295.092,-80.961,178.108,19.058,152.473
C03602=1096.509,295.339,-80.991,178.112,19.060,152.473
C03603=1096.514,295.588,-81.021,178.115,19.062,152.473
C03604=1096.520,295.836,-81.051,178.118,19.065,152.473
C03605=1096.526,296.083,-81.081,178.121,19.067,152.473
C03606=1096.532,296.332,-81.111,178.125,19.069,152.473
C03607=1096.537,296.580,-81.141,178.128,19.072,152.473
C03608=1096.543,296.828,-81.172,178.131,19.074,152.473
C03609=1096.549,297.076,-81.201,178.134,19.076,152.473
C03610=1096.555,297.324,-81.232,178.138,19.079,152.473
C03611=1096.560,297.572,-81.263,178.141,19.081,152.473
C03612=1096.565,297.820,-81.293,178.144,19.083,152.473
C03613=1096.571,298.068,-81.322,178.147,19.085,152.472
C03614=1096.577,298.316,-81.353,178.150,19.088,152.473
C03615=1096.583,298.564,-81.383,178.154,19.090,152.472
C03616=1096.588,298.812,-81.414,178.157,19.093,152.472
C03617=1096.594,299.060,-81.444,178.160,19.095,152.472
C03618=1096.599,299.308,-81.474,178.163,19.098,152.472
C03619=1096.604,299.556,-81.505,178.166,19.100,152.472
C03620=1096.610,299.804,-81.535,178.170,19.102,152.472
C03621=1096.616,300.052,-81.566,178.173,19.105,152.472
C03622=1096.621,300.300,-81.597,178.176,19.107,152.472
C03623=1096.627,300.548,-81.627,178.179,19.110,152.472
C03624=1096.632,300.796,-81.657,178.182,19.112,152.472
C03625=1096.638,301.044,-81.688,178.186,19.115,152.472
C03626=1096.644,301.292,-81.719,178.189,19.117,152.472
C03627=1096.650,301.540,-81.749,178.192,19.119,152.472
C03628=1096.655,301.788,-81.780,178.195,19.122,152.472
C03629=1096.661,302.036,-81.811,178.198,19.124,152.472
C03630=1096.666,302.284,-81.842,178.202,19.127,152.472
C03631=1096.675,302.670,-81.888,178.207,19.131,152.472
C03632=1096.684,303.056,-81.937,178.212,19.135,152.472
C03633=1096.692,303.443,-81.984,178.217,19.138,152.472
C03634=1096.701,303.829,-82.032,178.222,19.142,152.472
C03635=1096.706,304.077,-82.063,178.225,19.145,152.472
C03636=1096.712,304.325,-82.094,178.229,19.147,152.472
C03637=1096.717,304.573,-82.125,178.232,19.150,152.472
C03638=1096.723,304.821,-82.155,178.235,19.152,152.472
C03639=1096.729,305.068,-82.186,178.238,19.155,152.472
C03640=1096.734,305.317,-82.217,178.241,19.157,152.472
